LIN {X 0,Y 203.434,Z 438.559,A -85,B 0,C 180,E1 -21715.309,E2 -21715.309} C_VEL
LIN {X 0,Y 205.387,Z 432.116,A -85,B 0,C 180,E1 -21716.674,E2 -21716.674} C_VEL
LIN {X 0,Y 207.361,Z 424.448,A -85,B 0,C 180,E1 -21718.015,E2 -21718.015} C_VEL
LIN {X 0,Y 209.258,Z 416.269,A -85,B 0,C 180,E1 -21719.141,E2 -21719.141} C_VEL
LIN {X 0,Y 210.873,Z 408.266,A -85,B 0,C 180,E1 -21719.994,E2 -21719.994} C_VEL
LIN {X 0,Y 212.446,Z 398.341,A -85,B 0,C 180,E1 -21720.77,E2 -21720.77} C_VEL
LIN {X 0,Y 213.416,Z 388.623,A -85,B 0,C 180,E1 -21721.297,E2 -21721.297} C_VEL
LIN {X 0,Y 214.643,Z 363.756,A -85,B 0,C 180,E1 -21722.215,E2 -21722.215} C_VEL
LIN {X 0,Y 212.631,Z 347.83,A -85,B 0,C 180,E1 -21723.396,E2 -21723.396} C_VEL
LIN {X 0,Y 207.609,Z 336.115,A -85,B 0,C 180,E1 -21725.154,E2 -21725.154} C_VEL
LIN {X 0,Y 202.459,Z 325.893,A -85,B 0,C 180,E1 -21727.022,E2 -21727.022} C_VEL
LIN {X 0,Y 199.408,Z 320.617,A -85,B 0,C 180,E1 -21728.178,E2 -21728.178} C_VEL
LIN {X 0,Y 196.695,Z 316.069,A -85,B 0,C 180,E1 -21729.25,E2 -21729.25} C_VEL
LIN {X 0,Y 194.085,Z 311.74,A -85,B 0,C 180,E1 -21730.35,E2 -21730.35} C_VEL
LIN {X 0,Y 193.924,Z 311.308,A -85,B 0,C 180,E1 -21730.442,E2 -21730.442} C_VEL
LIN {X 0,Y 192.535,Z 306.316,A -85,B 0,C 180,E1 -21734.415,E2 -21734.415} C_VEL
LIN {X 0,Y 192.513,Z 306.314,A -85,B 0,C 180,E1 -21740.051,E2 -21740.051} C_VEL
LIN {X 0,Y 192.556,Z 306.307,A -85,B 0,C 180,E1 -21744.27,E2 -21744.27} C_VEL
LIN {X 0,Y 192.603,Z 306.292,A -85,B 0,C 180,E1 -21747.059,E2 -21747.059} C_VEL
LIN {X 0,Y 192.66,Z 306.284,A -85,B 0,C 180,E1 -21751.691,E2 -21751.691} C_VEL
LIN {X 0,Y 192.68,Z 306.291,A -85,B 0,C 180,E1 -21756.345,E2 -21756.345} C_VEL
LIN {X 0,Y 192.726,Z 306.291,A -85,B 0,C 180,E1 -21761.459,E2 -21761.459} C_VEL
LIN {X 0,Y 192.756,Z 306.268,A -85,B 0,C 180,E1 -21765.213,E2 -21765.213} C_VEL
LIN {X 0,Y 192.94,Z 306.247,A -85,B 0,C 180,E1 -21769.567,E2 -21769.567} C_VEL
LIN {X 0,Y 193.035,Z 306.233,A -85,B 0,C 180,E1 -21771.626,E2 -21771.626} C_VEL
LIN {X 0,Y 193.254,Z 306.208,A -85,B 0,C 180,E1 -21777.916,E2 -21777.916} C_VEL
LIN {X 0,Y 193.436,Z 306.199,A -85,B 0,C 180,E1 -21780,E2 -21780} C_VEL
LIN {X 0,Y 192.956,Z 306.254,A -85,B 0,C 180,E1 -21784.178,E2 -21784.178} C_VEL
LIN {X 0,Y 193.019,Z 306.241,A -85,B 0,C 180,E1 -21788.375,E2 -21788.375} C_VEL
LIN {X 0,Y 192.795,Z 306.27,A -85,B 0,C 180,E1 -21792.634,E2 -21792.634} C_VEL
LIN {X 0,Y 192.751,Z 306.28,A -85,B 0,C 180,E1 -21796.96,E2 -21796.96} C_VEL
LIN {X 0,Y 192.646,Z 306.299,A -85,B 0,C 180,E1 -21801.256,E2 -21801.256} C_VEL
LIN {X 0,Y 193.578,Z 309.046,A -85,B 0,C 180,E1 -21801.778,E2 -21801.778} C_VEL
LIN {X 0,Y 196.018,Z 311.688,A -85,B 0,C 180,E1 -21802.74,E2 -21802.74} C_VEL
LIN {X 0,Y 198.027,Z 314.946,A -85,B 0,C 180,E1 -21803.55,E2 -21803.55} C_VEL
LIN {X 0,Y 199.444,Z 316.867,A -85,B 0,C 180,E1 -21804.08,E2 -21804.08} C_VEL
LIN {X 0,Y 204.639,Z 324.932,A -85,B 0,C 180,E1 -21805.977,E2 -21805.977} C_VEL
LIN {X 0,Y 208.254,Z 331.276,A -85,B 0,C 180,E1 -21807.222,E2 -21807.222} C_VEL
LIN {X 0,Y 213.52,Z 342.533,A -85,B 0,C 180,E1 -21809.009,E2 -21809.009} C_VEL
LIN {X 0,Y 215.53,Z 347.517,A -85,B 0,C 180,E1 -21809.689,E2 -21809.689} C_VEL
LIN {X 0,Y 213.587,Z 380.961,A -85,B 0,C 180,E1 -21810.874,E2 -21810.874} C_VEL
LIN {X 0,Y 212.575,Z 391.195,A -85,B 0,C 180,E1 -21811.488,E2 -21811.488} C_VEL
LIN {X 0,Y 210.726,Z 403.434,A -85,B 0,C 180,E1 -21812.62,E2 -21812.62} C_VEL
LIN {X 0,Y 209.023,Z 411.772,A -85,B 0,C 180,E1 -21813.68,E2 -21813.68} C_VEL
LIN {X 0,Y 207.002,Z 419.999,A -85,B 0,C 180,E1 -21815.01,E2 -21815.01} C_VEL
LIN {X 0,Y 204.74,Z 428.007,A -85,B 0,C 180,E1 -21816.644,E2 -21816.644} C_VEL
LIN {X 0,Y 202.714,Z 434.266,A -85,B 0,C 180,E1 -21818.206,E2 -21818.206} C_VEL
LIN {X 0,Y 200.305,Z 440.944,A -85,B 0,C 180,E1 -21820.261,E2 -21820.261} C_VEL
LIN {X 0,Y 198.095,Z 446.483,A -85,B 0,C 180,E1 -21822.383,E2 -21822.383} C_VEL
LIN {X 0,Y 196.474,Z 450.562,A -85,B 0,C 180,E1 -21824.325,E2 -21824.325} C_VEL
LIN {X 0,Y 194.661,Z 454.577,A -85,B 0,C 180,E1 -21826.69,E2 -21826.69} C_VEL
LIN {X 0,Y 193.231,Z 457.717,A -85,B 0,C 180,E1 -21829.106,E2 -21829.106} C_VEL
LIN {X 0,Y 192.017,Z 460.05,A -85,B 0,C 180,E1 -21831.523,E2 -21831.523} C_VEL
LIN {X 0,Y 191.113,Z 461.68,A -85,B 0,C 180,E1 -21834.002,E2 -21834.002} C_VEL
LIN {X 0,Y 190.483,Z 462.591,A -85,B 0,C 180,E1 -21836.398,E2 -21836.398} C_VEL
LIN {X 0,Y 190.065,Z 462.86,A -85,B 0,C 180,E1 -21838.825,E2 -21838.825} C_VEL
LIN {X 0,Y 189.849,Z 462.453,A -85,B 0,C 180,E1 -21841.234,E2 -21841.234} C_VEL
LIN {X 0,Y 189.868,Z 461.377,A -85,B 0,C 180,E1 -21843.63,E2 -21843.63} C_VEL
LIN {X 0,Y 190.373,Z 458.386,A -85,B 0,C 180,E1 -21847.358,E2 -21847.358} C_VEL
LIN {X 0,Y 190.828,Z 455.896,A -85,B 0,C 180,E1 -21849.521,E2 -21849.521} C_VEL
LIN {X 0,Y 191.651,Z 451.34,A -85,B 0,C 180,E1 -21852.449,E2 -21852.449} C_VEL
LIN {X 0,Y 192.454,Z 447.029,A -85,B 0,C 180,E1 -21854.648,E2 -21854.648} C_VEL
LIN {X 0,Y 193.564,Z 441.616,A -85,B 0,C 180,E1 -21856.884,E2 -21856.884} C_VEL
LIN {X 0,Y 194.915,Z 434.909,A -85,B 0,C 180,E1 -21859.12,E2 -21859.12} C_VEL
LIN {X 0,Y 196.196,Z 428.057,A -85,B 0,C 180,E1 -21860.984,E2 -21860.984} C_VEL
LIN {X 0,Y 197.546,Z 420.587,A -85,B 0,C 180,E1 -21862.641,E2 -21862.641} C_VEL
LIN {X 0,Y 198.959,Z 412.007,A -85,B 0,C 180,E1 -21864.171,E2 -21864.171} C_VEL
LIN {X 0,Y 200.337,Z 401.733,A -85,B 0,C 180,E1 -21865.599,E2 -21865.599} C_VEL
LIN {X 0,Y 201.427,Z 390.601,A -85,B 0,C 180,E1 -21866.687,E2 -21866.687} C_VEL
LIN {X 0,Y 202.147,Z 380.872,A -85,B 0,C 180,E1 -21867.322,E2 -21867.322} C_VEL
LIN {X 0,Y 203.703,Z 338.888,A -85,B 0,C 180,E1 -21868.912,E2 -21868.912} C_VEL
LIN {X 0,Y 202.454,Z 331.462,A -85,B 0,C 180,E1 -21869.352,E2 -21869.352} C_VEL
LIN {X 0,Y 196.567,Z 313.956,A -85,B 0,C 180,E1 -21870.782,E2 -21870.782} C_VEL
LIN {X 0,Y 193.402,Z 306.719,A -85,B 0,C 180,E1 -21871.497,E2 -21871.497} C_VEL
LIN {X 0,Y 193.304,Z 306.221,A -85,B 0,C 180,E1 -21871.615,E2 -21871.615} C_VEL
LIN {X 0,Y 193.033,Z 306.255,A -85,B 0,C 180,E1 -21878.374,E2 -21878.374} C_VEL
LIN {X 0,Y 192.798,Z 306.271,A -85,B 0,C 180,E1 -21882.633,E2 -21882.633} C_VEL
LIN {X 0,Y 192.749,Z 306.286,A -85,B 0,C 180,E1 -21886.959,E2 -21886.959} C_VEL
LIN {X 0,Y 192.609,Z 306.28,A -85,B 0,C 180,E1 -21891.4,E2 -21891.4} C_VEL
LIN {X 0,Y 192.648,Z 306.291,A -85,B 0,C 180,E1 -21894.212,E2 -21894.212} C_VEL
LIN {X 0,Y 192.65,Z 306.305,A -85,B 0,C 180,E1 -21898.891,E2 -21898.891} C_VEL
LIN {X 0,Y 192.598,Z 306.3,A -85,B 0,C 180,E1 -21903.185,E2 -21903.185} C_VEL
LIN {X 0,Y 192.551,Z 306.312,A -85,B 0,C 180,E1 -21908.351,E2 -21908.351} C_VEL
LIN {X 0,Y 192.537,Z 306.306,A -85,B 0,C 180,E1 -21913.909,E2 -21913.909} C_VEL
LIN {X 0,Y 192.576,Z 306.308,A -85,B 0,C 180,E1 -21918.935,E2 -21918.935} C_VEL
LIN {X 0,Y 192.616,Z 306.291,A -85,B 0,C 180,E1 -21923.388,E2 -21923.388} C_VEL
LIN {X 0,Y 192.604,Z 306.294,A -85,B 0,C 180,E1 -21927.059,E2 -21927.059} C_VEL
LIN {X 0,Y 192.661,Z 306.298,A -85,B 0,C 180,E1 -21931.691,E2 -21931.691} C_VEL
LIN {X 0,Y 192.702,Z 306.283,A -85,B 0,C 180,E1 -21936.348,E2 -21936.348} C_VEL
LIN {X 0,Y 192.728,Z 306.276,A -85,B 0,C 180,E1 -21941.457,E2 -21941.457} C_VEL
LIN {X 0,Y 192.758,Z 306.285,A -85,B 0,C 180,E1 -21945.213,E2 -21945.213} C_VEL
LIN {X 0,Y 192.941,Z 306.26,A -85,B 0,C 180,E1 -21949.566,E2 -21949.566} C_VEL
LIN {X 0,Y 192.978,Z 306.24,A -85,B 0,C 180,E1 -21953.727,E2 -21953.727} C_VEL
LIN {X 0,Y 193.255,Z 306.214,A -85,B 0,C 180,E1 -21957.916,E2 -21957.916} C_VEL
LIN {X 0,Y 193.436,Z 306.198,A -85,B 0,C 180,E1 -21960,E2 -21960} C_VEL
LIN {X 0,Y 192.964,Z 306.258,A -85,B 0,C 180,E1 -21964.177,E2 -21964.177} C_VEL
LIN {X 0,Y 193.03,Z 306.237,A -85,B 0,C 180,E1 -21968.374,E2 -21968.374} C_VEL
LIN {X 0,Y 192.795,Z 306.275,A -85,B 0,C 180,E1 -21972.634,E2 -21972.634} C_VEL
LIN {X 0,Y 192.75,Z 306.286,A -85,B 0,C 180,E1 -21976.959,E2 -21976.959} C_VEL
LIN {X 0,Y 192.61,Z 306.292,A -85,B 0,C 180,E1 -21981.4,E2 -21981.4} C_VEL
LIN {X 0,Y 192.642,Z 306.3,A -85,B 0,C 180,E1 -21984.213,E2 -21984.213} C_VEL
LIN {X 0,Y 192.639,Z 306.296,A -85,B 0,C 180,E1 -21988.889,E2 -21988.889} C_VEL
LIN {X 0,Y 192.592,Z 306.307,A -85,B 0,C 180,E1 -21993.187,E2 -21993.187} C_VEL
LIN {X 0,Y 192.547,Z 306.303,A -85,B 0,C 180,E1 -21998.353,E2 -21998.353} C_VEL
LIN {X 0,Y 192.488,Z 306.311,A -85,B 0,C 180,E1 -22003.096,E2 -22003.096} C_VEL
LIN {X 0,Y 192.489,Z 306.32,A -85,B 0,C 180,E1 -22006.905,E2 -22006.905} C_VEL
LIN {X 0,Y 192.549,Z 306.312,A -85,B 0,C 180,E1 -22011.649,E2 -22011.649} C_VEL
LIN {X 0,Y 192.654,Z 306.48,A -85,B 0,C 180,E1 -22016.513,E2 -22016.513} C_VEL
LIN {X 0,Y 194.109,Z 313.398,A -85,B 0,C 180,E1 -22020.468,E2 -22020.468} C_VEL
LIN {X 0,Y 199.249,Z 328.764,A -85,B 0,C 180,E1 -22021.772,E2 -22021.772} C_VEL
LIN {X 0,Y 203.033,Z 359.935,A -85,B 0,C 180,E1 -22023.469,E2 -22023.469} C_VEL
LIN {X 0,Y 202.374,Z 380.986,A -85,B 0,C 180,E1 -22024.245,E2 -22024.245} C_VEL
LIN {X 0,Y 201.379,Z 386.811,A -85,B 0,C 180,E1 -22024.384,E2 -22024.384} C_VEL
LIN {X 0,Y 197.854,Z 396.121,A -85,B 0,C 180,E1 -22024.575,E2 -22024.575} C_VEL
LIN {X 0,Y 194.572,Z 404.335,A -85,B 0,C 180,E1 -22024.961,E2 -22024.961} C_VEL
LIN {X 0,Y 193.494,Z 408.938,A -85,B 0,C 180,E1 -22025.38,E2 -22025.38} C_VEL
LIN {X 0,Y 193.28,Z 410.781,A -85,B 0,C 180,E1 -22025.582,E2 -22025.582} C_VEL
LIN {X 0,Y 191.835,Z 421.682,A -85,B 0,C 180,E1 -22027.093,E2 -22027.093} C_VEL
LIN {X 0,Y 190.225,Z 430.12,A -85,B 0,C 180,E1 -22028.603,E2 -22028.603} C_VEL
LIN {X 0,Y 189.015,Z 437.111,A -85,B 0,C 180,E1 -22030.167,E2 -22030.167} C_VEL
LIN {X 0,Y 187.632,Z 443.888,A -85,B 0,C 180,E1 -22032.001,E2 -22032.001} C_VEL
LIN {X 0,Y 186.264,Z 450.309,A -85,B 0,C 180,E1 -22034.125,E2 -22034.125} C_VEL
LIN {X 0,Y 185.196,Z 455.643,A -85,B 0,C 180,E1 -22036.28,E2 -22036.28} C_VEL
LIN {X 0,Y 184.197,Z 461.047,A -85,B 0,C 180,E1 -22039.002,E2 -22039.002} C_VEL
LIN {X 0,Y 183.657,Z 464.529,A -85,B 0,C 180,E1 -22041.195,E2 -22041.195} C_VEL
LIN {X 0,Y 183.178,Z 468.522,A -85,B 0,C 180,E1 -22044.496,E2 -22044.496} C_VEL
LIN {X 0,Y 183.099,Z 471.231,A -85,B 0,C 180,E1 -22047.8,E2 -22047.8} C_VEL
LIN {X 0,Y 183.2,Z 472.28,A -85,B 0,C 180,E1 -22050,E2 -22050} C_VEL
LIN {X 0,Y 183.052,Z 472.991,A -85,B 0,C 180,E1 -22053.412,E2 -22053.412} C_VEL
LIN {X 0,Y 183.303,Z 472.546,A -85,B 0,C 180,E1 -22056.605,E2 -22056.605} C_VEL
LIN {X 0,Y 183.684,Z 471.57,A -85,B 0,C 180,E1 -22058.803,E2 -22058.803} C_VEL
LIN {X 0,Y 184.348,Z 470.105,A -85,B 0,C 180,E1 -22060.988,E2 -22060.988} C_VEL
LIN {X 0,Y 185.765,Z 466.977,A -85,B 0,C 180,E1 -22064.235,E2 -22064.235} C_VEL
LIN {X 0,Y 187.76,Z 462.559,A -85,B 0,C 180,E1 -22067.424,E2 -22067.424} C_VEL
LIN {X 0,Y 190.383,Z 456.487,A -85,B 0,C 180,E1 -22070.529,E2 -22070.529} C_VEL
LIN {X 0,Y 192.486,Z 451.491,A -85,B 0,C 180,E1 -22072.542,E2 -22072.542} C_VEL
LIN {X 0,Y 194.842,Z 445.491,A -85,B 0,C 180,E1 -22074.506,E2 -22074.506} C_VEL
LIN {X 0,Y 197.684,Z 437.209,A -85,B 0,C 180,E1 -22076.668,E2 -22076.668} C_VEL
LIN {X 0,Y 200.136,Z 429.569,A -85,B 0,C 180,E1 -22078.223,E2 -22078.223} C_VEL
LIN {X 0,Y 202.757,Z 419.419,A -85,B 0,C 180,E1 -22079.884,E2 -22079.884} C_VEL
LIN {X 0,Y 205.191,Z 408.083,A -85,B 0,C 180,E1 -22081.169,E2 -22081.169} C_VEL
LIN {X 0,Y 206.761,Z 398.675,A -85,B 0,C 180,E1 -22081.926,E2 -22081.926} C_VEL
LIN {X 0,Y 207.771,Z 389.397,A -85,B 0,C 180,E1 -22082.455,E2 -22082.455} C_VEL
LIN {X 0,Y 209.142,Z 364.971,A -85,B 0,C 180,E1 -22083.377,E2 -22083.377} C_VEL
LIN {X 0,Y 207.395,Z 350.739,A -85,B 0,C 180,E1 -22084.481,E2 -22084.481} C_VEL
LIN {X 0,Y 202.339,Z 338.752,A -85,B 0,C 180,E1 -22086.372,E2 -22086.372} C_VEL
LIN {X 0,Y 197.56,Z 329.355,A -85,B 0,C 180,E1 -22088.242,E2 -22088.242} C_VEL
LIN {X 0,Y 192.786,Z 321.063,A -85,B 0,C 180,E1 -22090.214,E2 -22090.214} C_VEL
LIN {X 0,Y 189.733,Z 316.142,A -85,B 0,C 180,E1 -22091.572,E2 -22091.572} C_VEL
LIN {X 0,Y 186.926,Z 311.969,A -85,B 0,C 180,E1 -22092.874,E2 -22092.874} C_VEL
LIN {X 0,Y 186.457,Z 310.795,A -85,B 0,C 180,E1 -22093.256,E2 -22093.256} C_VEL
LIN {X 0,Y 185.446,Z 307.2,A -85,B 0,C 180,E1 -22096.504,E2 -22096.504} C_VEL
LIN {X 0,Y 185.463,Z 307.191,A -85,B 0,C 180,E1 -22099.894,E2 -22099.894} C_VEL
LIN {X 0,Y 185.502,Z 307.179,A -85,B 0,C 180,E1 -22102.711,E2 -22102.711} C_VEL
LIN {X 0,Y 185.539,Z 307.172,A -85,B 0,C 180,E1 -22107.974,E2 -22107.974} C_VEL
LIN {X 0,Y 185.577,Z 307.178,A -85,B 0,C 180,E1 -22110.576,E2 -22110.576} C_VEL
LIN {X 0,Y 185.575,Z 307.181,A -85,B 0,C 180,E1 -22115.381,E2 -22115.381} C_VEL
LIN {X 0,Y 185.668,Z 307.17,A -85,B 0,C 180,E1 -22121.135,E2 -22121.135} C_VEL
LIN {X 0,Y 185.688,Z 307.146,A -85,B 0,C 180,E1 -22124.637,E2 -22124.637} C_VEL
LIN {X 0,Y 185.884,Z 307.126,A -85,B 0,C 180,E1 -22129.417,E2 -22129.417} C_VEL
LIN {X 0,Y 185.944,Z 307.133,A -85,B 0,C 180,E1 -22133.49,E2 -22133.49} C_VEL
LIN {X 0,Y 186.198,Z 307.086,A -85,B 0,C 180,E1 -22137.837,E2 -22137.837} C_VEL
LIN {X 0,Y 186.399,Z 307.076,A -85,B 0,C 180,E1 -22140,E2 -22140} C_VEL
LIN {X 0,Y 185.903,Z 307.134,A -85,B 0,C 180,E1 -22144.337,E2 -22144.337} C_VEL
LIN {X 0,Y 185.968,Z 307.12,A -85,B 0,C 180,E1 -22148.695,E2 -22148.695} C_VEL
LIN {X 0,Y 185.722,Z 307.152,A -85,B 0,C 180,E1 -22153.124,E2 -22153.124} C_VEL
LIN {X 0,Y 185.689,Z 307.236,A -85,B 0,C 180,E1 -22158.793,E2 -22158.793} C_VEL
LIN {X 0,Y 186.476,Z 309.725,A -85,B 0,C 180,E1 -22159.265,E2 -22159.265} C_VEL
LIN {X 0,Y 188.492,Z 312.038,A -85,B 0,C 180,E1 -22160.175,E2 -22160.175} C_VEL
LIN {X 0,Y 189.26,Z 312.966,A -85,B 0,C 180,E1 -22160.515,E2 -22160.515} C_VEL
LIN {X 0,Y 191.39,Z 316.203,A -85,B 0,C 180,E1 -22161.473,E2 -22161.473} C_VEL
LIN {X 0,Y 192.579,Z 317.611,A -85,B 0,C 180,E1 -22161.967,E2 -22161.967} C_VEL
LIN {X 0,Y 198.035,Z 325.775,A -85,B 0,C 180,E1 -22164.157,E2 -22164.157} C_VEL
LIN {X 0,Y 202.881,Z 333.982,A -85,B 0,C 180,E1 -22165.978,E2 -22165.978} C_VEL
LIN {X 0,Y 207.643,Z 343.937,A -85,B 0,C 180,E1 -22167.699,E2 -22167.699} C_VEL
LIN {X 0,Y 209.982,Z 349.731,A -85,B 0,C 180,E1 -22168.539,E2 -22168.539} C_VEL
LIN {X 0,Y 208.007,Z 381.708,A -85,B 0,C 180,E1 -22169.704,E2 -22169.704} C_VEL
LIN {X 0,Y 206.773,Z 392.837,A -85,B 0,C 180,E1 -22170.398,E2 -22170.398} C_VEL
LIN {X 0,Y 204.99,Z 403.83,A -85,B 0,C 180,E1 -22171.482,E2 -22171.482} C_VEL
LIN {X 0,Y 203.224,Z 412.033,A -85,B 0,C 180,E1 -22172.55,E2 -22172.55} C_VEL
LIN {X 0,Y 200.862,Z 420.979,A -85,B 0,C 180,E1 -22174.044,E2 -22174.044} C_VEL
LIN {X 0,Y 198.724,Z 428.205,A -85,B 0,C 180,E1 -22175.572,E2 -22175.572} C_VEL
LIN {X 0,Y 196.122,Z 435.719,A -85,B 0,C 180,E1 -22177.531,E2 -22177.531} C_VEL
LIN {X 0,Y 193.702,Z 441.948,A -85,B 0,C 180,E1 -22179.558,E2 -22179.558} C_VEL
LIN {X 0,Y 190.717,Z 449.06,A -85,B 0,C 180,E1 -22182.525,E2 -22182.525} C_VEL
LIN {X 0,Y 188.712,Z 453.553,A -85,B 0,C 180,E1 -22185.04,E2 -22185.04} C_VEL
LIN {X 0,Y 187.023,Z 456.907,A -85,B 0,C 180,E1 -22187.438,E2 -22187.438} C_VEL
LIN {X 0,Y 185.64,Z 459.533,A -85,B 0,C 180,E1 -22189.941,E2 -22189.941} C_VEL
LIN {X 0,Y 184.259,Z 461.783,A -85,B 0,C 180,E1 -22193.224,E2 -22193.224} C_VEL
LIN {X 0,Y 183.703,Z 462.53,A -85,B 0,C 180,E1 -22194.981,E2 -22194.981} C_VEL
LIN {X 0,Y 183.15,Z 463.007,A -85,B 0,C 180,E1 -22197.587,E2 -22197.587} C_VEL
LIN {X 0,Y 182.842,Z 462.818,A -85,B 0,C 180,E1 -22200.022,E2 -22200.022} C_VEL
LIN {X 0,Y 182.759,Z 462.008,A -85,B 0,C 180,E1 -22202.52,E2 -22202.52} C_VEL
LIN {X 0,Y 182.882,Z 460.569,A -85,B 0,C 180,E1 -22204.994,E2 -22204.994} C_VEL
LIN {X 0,Y 183.297,Z 458.47,A -85,B 0,C 180,E1 -22207.455,E2 -22207.455} C_VEL
LIN {X 0,Y 183.812,Z 455.703,A -85,B 0,C 180,E1 -22209.873,E2 -22209.873} C_VEL
LIN {X 0,Y 184.666,Z 451.157,A -85,B 0,C 180,E1 -22212.846,E2 -22212.846} C_VEL
LIN {X 0,Y 185.52,Z 446.633,A -85,B 0,C 180,E1 -22215.185,E2 -22215.185} C_VEL
LIN {X 0,Y 186.924,Z 440.18,A -85,B 0,C 180,E1 -22217.838,E2 -22217.838} C_VEL
LIN {X 0,Y 188.118,Z 434.356,A -85,B 0,C 180,E1 -22219.779,E2 -22219.779} C_VEL
LIN {X 0,Y 189.743,Z 426.108,A -85,B 0,C 180,E1 -22222.017,E2 -22222.017} C_VEL
LIN {X 0,Y 191.66,Z 415.505,A -85,B 0,C 180,E1 -22224.213,E2 -22224.213} C_VEL
LIN {X 0,Y 192.934,Z 407.016,A -85,B 0,C 180,E1 -22225.561,E2 -22225.561} C_VEL
LIN {X 0,Y 193.927,Z 398.525,A -85,B 0,C 180,E1 -22226.624,E2 -22226.624} C_VEL
LIN {X 0,Y 194.881,Z 389.268,A -85,B 0,C 180,E1 -22227.481,E2 -22227.481} C_VEL
LIN {X 0,Y 195.524,Z 379.672,A -85,B 0,C 180,E1 -22228.095,E2 -22228.095} C_VEL
LIN {X 0,Y 197.062,Z 339.354,A -85,B 0,C 180,E1 -22229.655,E2 -22229.655} C_VEL
LIN {X 0,Y 195.953,Z 333.197,A -85,B 0,C 180,E1 -22230.048,E2 -22230.048} C_VEL
LIN {X 0,Y 190.398,Z 316.71,A -85,B 0,C 180,E1 -22231.457,E2 -22231.457} C_VEL
LIN {X 0,Y 186.2,Z 307.493,A -85,B 0,C 180,E1 -22232.434,E2 -22232.434} C_VEL
LIN {X 0,Y 186.119,Z 307.113,A -85,B 0,C 180,E1 -22232.57,E2 -22232.57} C_VEL
LIN {X 0,Y 185.981,Z 307.132,A -85,B 0,C 180,E1 -22238.694,E2 -22238.694} C_VEL
LIN {X 0,Y 185.725,Z 307.153,A -85,B 0,C 180,E1 -22243.123,E2 -22243.123} C_VEL
LIN {X 0,Y 185.685,Z 307.165,A -85,B 0,C 180,E1 -22247.625,E2 -22247.625} C_VEL
LIN {X 0,Y 185.574,Z 307.156,A -85,B 0,C 180,E1 -22252.254,E2 -22252.254} C_VEL
LIN {X 0,Y 185.561,Z 307.187,A -85,B 0,C 180,E1 -22257.031,E2 -22257.031} C_VEL
LIN {X 0,Y 185.579,Z 307.183,A -85,B 0,C 180,E1 -22259.492,E2 -22259.492} C_VEL
LIN {X 0,Y 185.499,Z 307.187,A -85,B 0,C 180,E1 -22264.631,E2 -22264.631} C_VEL
LIN {X 0,Y 185.505,Z 307.193,A -85,B 0,C 180,E1 -22267.312,E2 -22267.312} C_VEL
LIN {X 0,Y 185.473,Z 307.189,A -85,B 0,C 180,E1 -22270.725,E2 -22270.725} C_VEL
LIN {X 0,Y 185.528,Z 307.185,A -85,B 0,C 180,E1 -22276.031,E2 -22276.031} C_VEL
LIN {X 0,Y 185.536,Z 307.184,A -85,B 0,C 180,E1 -22279.913,E2 -22279.913} C_VEL
LIN {X 0,Y 185.557,Z 307.172,A -85,B 0,C 180,E1 -22282.699,E2 -22282.699} C_VEL
LIN {X 0,Y 185.542,Z 307.178,A -85,B 0,C 180,E1 -22287.974,E2 -22287.974} C_VEL
LIN {X 0,Y 185.579,Z 307.179,A -85,B 0,C 180,E1 -22290.575,E2 -22290.575} C_VEL
LIN {X 0,Y 185.583,Z 307.173,A -85,B 0,C 180,E1 -22295.382,E2 -22295.382} C_VEL
LIN {X 0,Y 185.671,Z 307.155,A -85,B 0,C 180,E1 -22301.133,E2 -22301.133} C_VEL
LIN {X 0,Y 185.689,Z 307.165,A -85,B 0,C 180,E1 -22304.636,E2 -22304.636} C_VEL
LIN {X 0,Y 185.884,Z 307.139,A -85,B 0,C 180,E1 -22309.417,E2 -22309.417} C_VEL
LIN {X 0,Y 185.941,Z 307.116,A -85,B 0,C 180,E1 -22313.489,E2 -22313.489} C_VEL
LIN {X 0,Y 186.199,Z 307.093,A -85,B 0,C 180,E1 -22317.837,E2 -22317.837} C_VEL
LIN {X 0,Y 186.4,Z 307.074,A -85,B 0,C 180,E1 -22320,E2 -22320} C_VEL
LIN {X 0,Y 185.911,Z 307.136,A -85,B 0,C 180,E1 -22324.336,E2 -22324.336} C_VEL
LIN {X 0,Y 185.977,Z 307.115,A -85,B 0,C 180,E1 -22328.694,E2 -22328.694} C_VEL
LIN {X 0,Y 185.723,Z 307.157,A -85,B 0,C 180,E1 -22333.123,E2 -22333.123} C_VEL
LIN {X 0,Y 185.683,Z 307.167,A -85,B 0,C 180,E1 -22337.625,E2 -22337.625} C_VEL
LIN {X 0,Y 185.572,Z 307.172,A -85,B 0,C 180,E1 -22342.254,E2 -22342.254} C_VEL
LIN {X 0,Y 185.554,Z 307.183,A -85,B 0,C 180,E1 -22347.033,E2 -22347.033} C_VEL
LIN {X 0,Y 185.573,Z 307.177,A -85,B 0,C 180,E1 -22349.494,E2 -22349.494} C_VEL
LIN {X 0,Y 185.495,Z 307.193,A -85,B 0,C 180,E1 -22354.633,E2 -22354.633} C_VEL
LIN {X 0,Y 185.502,Z 307.186,A -85,B 0,C 180,E1 -22357.314,E2 -22357.314} C_VEL
LIN {X 0,Y 185.467,Z 307.173,A -85,B 0,C 180,E1 -22360.725,E2 -22360.725} C_VEL
LIN {X 0,Y 185.458,Z 307.195,A -85,B 0,C 180,E1 -22366.055,E2 -22366.055} C_VEL
LIN {X 0,Y 185.465,Z 307.194,A -85,B 0,C 180,E1 -22369.896,E2 -22369.896} C_VEL
LIN {X 0,Y 185.504,Z 307.188,A -85,B 0,C 180,E1 -22372.712,E2 -22372.712} C_VEL
LIN {X 0,Y 185.599,Z 307.344,A -85,B 0,C 180,E1 -22376.001,E2 -22376.001} C_VEL
LIN {X 0,Y 186.818,Z 313.253,A -85,B 0,C 180,E1 -22379.525,E2 -22379.525} C_VEL
LIN {X 0,Y 192.764,Z 330.38,A -85,B 0,C 180,E1 -22381.047,E2 -22381.047} C_VEL
LIN {X 0,Y 196.469,Z 361.488,A -85,B 0,C 180,E1 -22382.81,E2 -22382.81} C_VEL
LIN {X 0,Y 195.25,Z 390.957,A -85,B 0,C 180,E1 -22383.972,E2 -22383.972} C_VEL
LIN {X 0,Y 194.486,Z 400.625,A -85,B 0,C 180,E1 -22384.609,E2 -22384.609} C_VEL
LIN {X 0,Y 193.28,Z 410.781,A -85,B 0,C 180,E1 -22385.582,E2 -22385.582} C_VEL
LIN {X 0,Y 192.111,Z 416.18,A -85,B 0,C 180,E1 -22386.193,E2 -22386.193} C_VEL
LIN {X 0,Y 189.902,Z 421.303,A -85,B 0,C 180,E1 -22386.805,E2 -22386.805} C_VEL
LIN {X 0,Y 184.59,Z 430.867,A -85,B 0,C 180,E1 -22388.279,E2 -22388.279} C_VEL
LIN {X 0,Y 182.575,Z 435.503,A -85,B 0,C 180,E1 -22389.268,E2 -22389.268} C_VEL
LIN {X 0,Y 182.148,Z 436.983,A -85,B 0,C 180,E1 -22389.647,E2 -22389.647} C_VEL
LIN {X 0,Y 180.875,Z 442.987,A -85,B 0,C 180,E1 -22391.304,E2 -22391.304} C_VEL
LIN {X 0,Y 179.428,Z 449.523,A -85,B 0,C 180,E1 -22393.503,E2 -22393.503} C_VEL
LIN {X 0,Y 178.292,Z 454.958,A -85,B 0,C 180,E1 -22395.738,E2 -22395.738} C_VEL
LIN {X 0,Y 177.209,Z 460.451,A -85,B 0,C 180,E1 -22398.563,E2 -22398.563} C_VEL
LIN {X 0,Y 176.627,Z 464.014,A -85,B 0,C 180,E1 -22400.842,E2 -22400.842} C_VEL
LIN {X 0,Y 176.11,Z 468.082,A -85,B 0,C 180,E1 -22404.274,E2 -22404.274} C_VEL
LIN {X 0,Y 175.989,Z 470.154,A -85,B 0,C 180,E1 -22406.709,E2 -22406.709} C_VEL
LIN {X 0,Y 176.105,Z 471.979,A -85,B 0,C 180,E1 -22410,E2 -22410} C_VEL
LIN {X 0,Y 175.953,Z 472.7,A -85,B 0,C 180,E1 -22413.077,E2 -22413.077} C_VEL
LIN {X 0,Y 176.243,Z 472.404,A -85,B 0,C 180,E1 -22416.87,E2 -22416.87} C_VEL
LIN {X 0,Y 176.657,Z 471.477,A -85,B 0,C 180,E1 -22419.156,E2 -22419.156} C_VEL
LIN {X 0,Y 177.361,Z 470.084,A -85,B 0,C 180,E1 -22421.427,E2 -22421.427} C_VEL
LIN {X 0,Y 178.889,Z 467.03,A -85,B 0,C 180,E1 -22424.795,E2 -22424.795} C_VEL
LIN {X 0,Y 180.989,Z 462.721,A -85,B 0,C 180,E1 -22428.098,E2 -22428.098} C_VEL
LIN {X 0,Y 183.765,Z 456.804,A -85,B 0,C 180,E1 -22431.304,E2 -22431.304} C_VEL
LIN {X 0,Y 186.511,Z 450.517,A -85,B 0,C 180,E1 -22433.895,E2 -22433.895} C_VEL
LIN {X 0,Y 189.085,Z 444.378,A -85,B 0,C 180,E1 -22435.895,E2 -22435.895} C_VEL
LIN {X 0,Y 191.416,Z 437.969,A -85,B 0,C 180,E1 -22437.615,E2 -22437.615} C_VEL
LIN {X 0,Y 194.289,Z 429.425,A -85,B 0,C 180,E1 -22439.426,E2 -22439.426} C_VEL
LIN {X 0,Y 196.695,Z 420.661,A -85,B 0,C 180,E1 -22440.904,E2 -22440.904} C_VEL
LIN {X 0,Y 199.465,Z 408.835,A -85,B 0,C 180,E1 -22442.336,E2 -22442.336} C_VEL
LIN {X 0,Y 201.227,Z 398.833,A -85,B 0,C 180,E1 -22443.166,E2 -22443.166} C_VEL
LIN {X 0,Y 202.264,Z 389.942,A -85,B 0,C 180,E1 -22443.694,E2 -22443.694} C_VEL
LIN {X 0,Y 203.687,Z 365.642,A -85,B 0,C 180,E1 -22444.644,E2 -22444.644} C_VEL
LIN {X 0,Y 202.263,Z 353.686,A -85,B 0,C 180,E1 -22445.614,E2 -22445.614} C_VEL
LIN {X 0,Y 197.931,Z 343.059,A -85,B 0,C 180,E1 -22447.372,E2 -22447.372} C_VEL
LIN {X 0,Y 192.277,Z 331.715,A -85,B 0,C 180,E1 -22449.74,E2 -22449.74} C_VEL
LIN {X 0,Y 188.721,Z 325.73,A -85,B 0,C 180,E1 -22451.326,E2 -22451.326} C_VEL
LIN {X 0,Y 185.913,Z 321.155,A -85,B 0,C 180,E1 -22452.653,E2 -22452.653} C_VEL
LIN {X 0,Y 182.488,Z 315.869,A -85,B 0,C 180,E1 -22454.367,E2 -22454.367} C_VEL
LIN {X 0,Y 179.527,Z 311.542,A -85,B 0,C 180,E1 -22455.984,E2 -22455.984} C_VEL
LIN {X 0,Y 179.104,Z 310.487,A -85,B 0,C 180,E1 -22456.34,E2 -22456.34} C_VEL
LIN {X 0,Y 178.421,Z 308.065,A -85,B 0,C 180,E1 -22458.865,E2 -22458.865} C_VEL
LIN {X 0,Y 178.418,Z 308.064,A -85,B 0,C 180,E1 -22463.782,E2 -22463.782} C_VEL
LIN {X 0,Y 178.481,Z 308.053,A -85,B 0,C 180,E1 -22466.546,E2 -22466.546} C_VEL
LIN {X 0,Y 178.518,Z 308.061,A -85,B 0,C 180,E1 -22470.006,E2 -22470.006} C_VEL
LIN {X 0,Y 178.515,Z 308.058,A -85,B 0,C 180,E1 -22474.886,E2 -22474.886} C_VEL
LIN {X 0,Y 178.616,Z 308.046,A -85,B 0,C 180,E1 -22480.786,E2 -22480.786} C_VEL
LIN {X 0,Y 178.651,Z 308.034,A -85,B 0,C 180,E1 -22486.348,E2 -22486.348} C_VEL
LIN {X 0,Y 178.908,Z 307.989,A -85,B 0,C 180,E1 -22490.96,E2 -22490.96} C_VEL
LIN {X 0,Y 178.858,Z 308,A -85,B 0,C 180,E1 -22495.493,E2 -22495.493} C_VEL
LIN {X 0,Y 179.363,Z 307.952,A -85,B 0,C 180,E1 -22500,E2 -22500} C_VEL
LIN {X 0,Y 178.85,Z 308.014,A -85,B 0,C 180,E1 -22504.508,E2 -22504.508} C_VEL
LIN {X 0,Y 178.899,Z 308.003,A -85,B 0,C 180,E1 -22509.041,E2 -22509.041} C_VEL
LIN {X 0,Y 178.633,Z 308.049,A -85,B 0,C 180,E1 -22514.817,E2 -22514.817} C_VEL
LIN {X 0,Y 178.625,Z 308.042,A -85,B 0,C 180,E1 -22515.767,E2 -22515.767} C_VEL
LIN {X 0,Y 179.529,Z 310.76,A -85,B 0,C 180,E1 -22516.415,E2 -22516.415} C_VEL
LIN {X 0,Y 181.521,Z 312.92,A -85,B 0,C 180,E1 -22517.461,E2 -22517.461} C_VEL
LIN {X 0,Y 182.387,Z 313.597,A -85,B 0,C 180,E1 -22517.883,E2 -22517.883} C_VEL
LIN {X 0,Y 184.268,Z 316.842,A -85,B 0,C 180,E1 -22518.883,E2 -22518.883} C_VEL
LIN {X 0,Y 185.987,Z 318.787,A -85,B 0,C 180,E1 -22519.679,E2 -22519.679} C_VEL
LIN {X 0,Y 188.59,Z 322.441,A -85,B 0,C 180,E1 -22520.877,E2 -22520.877} C_VEL
LIN {X 0,Y 194.026,Z 330.695,A -85,B 0,C 180,E1 -22523.216,E2 -22523.216} C_VEL
LIN {X 0,Y 198.595,Z 338.507,A -85,B 0,C 180,E1 -22525.025,E2 -22525.025} C_VEL
LIN {X 0,Y 203.38,Z 349.007,A -85,B 0,C 180,E1 -22526.893,E2 -22526.893} C_VEL
LIN {X 0,Y 204.511,Z 351.786,A -85,B 0,C 180,E1 -22527.32,E2 -22527.32} C_VEL
LIN {X 0,Y 202.578,Z 381.818,A -85,B 0,C 180,E1 -22528.438,E2 -22528.438} C_VEL
LIN {X 0,Y 201.319,Z 392.753,A -85,B 0,C 180,E1 -22529.128,E2 -22529.128} C_VEL
LIN {X 0,Y 199.348,Z 404.198,A -85,B 0,C 180,E1 -22530.263,E2 -22530.263} C_VEL
LIN {X 0,Y 197.187,Z 413.568,A -85,B 0,C 180,E1 -22531.539,E2 -22531.539} C_VEL
LIN {X 0,Y 194.993,Z 421.421,A -85,B 0,C 180,E1 -22532.9,E2 -22532.9} C_VEL
LIN {X 0,Y 192.776,Z 428.493,A -85,B 0,C 180,E1 -22534.431,E2 -22534.431} C_VEL
LIN {X 0,Y 190.293,Z 435.277,A -85,B 0,C 180,E1 -22536.223,E2 -22536.223} C_VEL
LIN {X 0,Y 187.804,Z 441.351,A -85,B 0,C 180,E1 -22538.202,E2 -22538.202} C_VEL
LIN {X 0,Y 185.165,Z 447.263,A -85,B 0,C 180,E1 -22540.617,E2 -22540.617} C_VEL
LIN {X 0,Y 182.318,Z 453.436,A -85,B 0,C 180,E1 -22543.937,E2 -22543.937} C_VEL
LIN {X 0,Y 180.134,Z 457.442,A -85,B 0,C 180,E1 -22546.943,E2 -22546.943} C_VEL
LIN {X 0,Y 178.69,Z 459.986,A -85,B 0,C 180,E1 -22549.539,E2 -22549.539} C_VEL
LIN {X 0,Y 177.049,Z 462.328,A -85,B 0,C 180,E1 -22553.458,E2 -22553.458} C_VEL
LIN {X 0,Y 176.165,Z 463.178,A -85,B 0,C 180,E1 -22556.907,E2 -22556.907} C_VEL
LIN {X 0,Y 175.867,Z 463.173,A -85,B 0,C 180,E1 -22558.702,E2 -22558.702} C_VEL
LIN {X 0,Y 175.68,Z 462.484,A -85,B 0,C 180,E1 -22561.655,E2 -22561.655} C_VEL
LIN {X 0,Y 175.688,Z 461.458,A -85,B 0,C 180,E1 -22563.895,E2 -22563.895} C_VEL
LIN {X 0,Y 176.039,Z 459.424,A -85,B 0,C 180,E1 -22566.669,E2 -22566.669} C_VEL
LIN {X 0,Y 176.789,Z 455.481,A -85,B 0,C 180,E1 -22570.251,E2 -22570.251} C_VEL
LIN {X 0,Y 177.586,Z 451.383,A -85,B 0,C 180,E1 -22573.017,E2 -22573.017} C_VEL
LIN {X 0,Y 178.624,Z 446.193,A -85,B 0,C 180,E1 -22575.765,E2 -22575.765} C_VEL
LIN {X 0,Y 180.01,Z 440.132,A -85,B 0,C 180,E1 -22578.313,E2 -22578.313} C_VEL
LIN {X 0,Y 181.372,Z 433.644,A -85,B 0,C 180,E1 -22580.521,E2 -22580.521} C_VEL
LIN {X 0,Y 183.126,Z 425.198,A -85,B 0,C 180,E1 -22582.835,E2 -22582.835} C_VEL
LIN {X 0,Y 184.86,Z 415.667,A -85,B 0,C 180,E1 -22584.832,E2 -22584.832} C_VEL
LIN {X 0,Y 186.19,Z 407.246,A -85,B 0,C 180,E1 -22586.213,E2 -22586.213} C_VEL
LIN {X 0,Y 187.224,Z 398.769,A -85,B 0,C 180,E1 -22587.311,E2 -22587.311} C_VEL
LIN {X 0,Y 188.226,Z 389.111,A -85,B 0,C 180,E1 -22588.231,E2 -22588.231} C_VEL
LIN {X 0,Y 188.869,Z 380.199,A -85,B 0,C 180,E1 -22588.817,E2 -22588.817} C_VEL
LIN {X 0,Y 190.475,Z 339.977,A -85,B 0,C 180,E1 -22590.43,E2 -22590.43} C_VEL
LIN {X 0,Y 189.586,Z 335.354,A -85,B 0,C 180,E1 -22590.743,E2 -22590.743} C_VEL
LIN {X 0,Y 184.378,Z 319.805,A -85,B 0,C 180,E1 -22592.128,E2 -22592.128} C_VEL
LIN {X 0,Y 179.196,Z 309.041,A -85,B 0,C 180,E1 -22593.373,E2 -22593.373} C_VEL
LIN {X 0,Y 178.971,Z 308.004,A -85,B 0,C 180,E1 -22593.489,E2 -22593.489} C_VEL
LIN {X 0,Y 178.91,Z 308.012,A -85,B 0,C 180,E1 -22599.04,E2 -22599.04} C_VEL
LIN {X 0,Y 178.653,Z 308.036,A -85,B 0,C 180,E1 -22603.652,E2 -22603.652} C_VEL
LIN {X 0,Y 178.61,Z 308.038,A -85,B 0,C 180,E1 -22609.202,E2 -22609.202} C_VEL
LIN {X 0,Y 178.52,Z 308.056,A -85,B 0,C 180,E1 -22615.113,E2 -22615.113} C_VEL
LIN {X 0,Y 178.501,Z 308.062,A -85,B 0,C 180,E1 -22620.785,E2 -22620.785} C_VEL
LIN {X 0,Y 178.485,Z 308.06,A -85,B 0,C 180,E1 -22624.218,E2 -22624.218} C_VEL
LIN {X 0,Y 178.396,Z 308.075,A -85,B 0,C 180,E1 -22629.073,E2 -22629.073} C_VEL
LIN {X 0,Y 178.413,Z 308.058,A -85,B 0,C 180,E1 -22632.039,E2 -22632.039} C_VEL
LIN {X 0,Y 178.442,Z 308.063,A -85,B 0,C 180,E1 -22635.147,E2 -22635.147} C_VEL
LIN {X 0,Y 178.48,Z 308.064,A -85,B 0,C 180,E1 -22638.429,E2 -22638.429} C_VEL
LIN {X 0,Y 178.457,Z 308.049,A -85,B 0,C 180,E1 -22643.791,E2 -22643.791} C_VEL
LIN {X 0,Y 178.488,Z 308.051,A -85,B 0,C 180,E1 -22646.547,E2 -22646.547} C_VEL
LIN {X 0,Y 178.52,Z 308.058,A -85,B 0,C 180,E1 -22650.005,E2 -22650.005} C_VEL
LIN {X 0,Y 178.521,Z 308.053,A -85,B 0,C 180,E1 -22654.882,E2 -22654.882} C_VEL
LIN {X 0,Y 178.619,Z 308.028,A -85,B 0,C 180,E1 -22660.784,E2 -22660.784} C_VEL
LIN {X 0,Y 178.652,Z 308.043,A -85,B 0,C 180,E1 -22666.347,E2 -22666.347} C_VEL
LIN {X 0,Y 178.906,Z 308.004,A -85,B 0,C 180,E1 -22670.959,E2 -22670.959} C_VEL
LIN {X 0,Y 179.145,Z 307.972,A -85,B 0,C 180,E1 -22677.751,E2 -22677.751} C_VEL
LIN {X 0,Y 179.363,Z 307.95,A -85,B 0,C 180,E1 -22680,E2 -22680} C_VEL
LIN {X 0,Y 178.859,Z 308.015,A -85,B 0,C 180,E1 -22684.507,E2 -22684.507} C_VEL
LIN {X 0,Y 178.906,Z 307.993,A -85,B 0,C 180,E1 -22689.04,E2 -22689.04} C_VEL
LIN {X 0,Y 178.651,Z 308.041,A -85,B 0,C 180,E1 -22693.652,E2 -22693.652} C_VEL
LIN {X 0,Y 178.616,Z 308.043,A -85,B 0,C 180,E1 -22699.214,E2 -22699.214} C_VEL
LIN {X 0,Y 178.515,Z 308.059,A -85,B 0,C 180,E1 -22705.114,E2 -22705.114} C_VEL
LIN {X 0,Y 178.517,Z 308.053,A -85,B 0,C 180,E1 -22709.993,E2 -22709.993} C_VEL
LIN {X 0,Y 178.48,Z 308.068,A -85,B 0,C 180,E1 -22714.219,E2 -22714.219} C_VEL
LIN {X 0,Y 178.391,Z 308.061,A -85,B 0,C 180,E1 -22719.075,E2 -22719.075} C_VEL
LIN {X 0,Y 178.395,Z 308.057,A -85,B 0,C 180,E1 -22722.046,E2 -22722.046} C_VEL
LIN {X 0,Y 178.391,Z 308.076,A -85,B 0,C 180,E1 -22725.164,E2 -22725.164} C_VEL
LIN {X 0,Y 178.401,Z 308.075,A -85,B 0,C 180,E1 -22728.46,E2 -22728.46} C_VEL
LIN {X 0,Y 178.433,Z 308.07,A -85,B 0,C 180,E1 -22733.787,E2 -22733.787} C_VEL
LIN {X 0,Y 178.507,Z 308.176,A -85,B 0,C 180,E1 -22735.423,E2 -22735.423} C_VEL
LIN {X 0,Y 179.566,Z 313.09,A -85,B 0,C 180,E1 -22738.478,E2 -22738.478} C_VEL
LIN {X 0,Y 185.825,Z 330.718,A -85,B 0,C 180,E1 -22740.17,E2 -22740.17} C_VEL
LIN {X 0,Y 186.958,Z 336.463,A -85,B 0,C 180,E1 -22740.575,E2 -22740.575} C_VEL
LIN {X 0,Y 189.858,Z 362.19,A -85,B 0,C 180,E1 -22742.063,E2 -22742.063} C_VEL
LIN {X 0,Y 188.572,Z 391.605,A -85,B 0,C 180,E1 -22743.271,E2 -22743.271} C_VEL
LIN {X 0,Y 187.561,Z 402.609,A -85,B 0,C 180,E1 -22744.051,E2 -22744.051} C_VEL
LIN {X 0,Y 186.227,Z 413.338,A -85,B 0,C 180,E1 -22745.243,E2 -22745.243} C_VEL
LIN {X 0,Y 184.732,Z 423.256,A -85,B 0,C 180,E1 -22746.753,E2 -22746.753} C_VEL
LIN {X 0,Y 183.104,Z 431.375,A -85,B 0,C 180,E1 -22748.32,E2 -22748.32} C_VEL
LIN {X 0,Y 182.148,Z 436.983,A -85,B 0,C 180,E1 -22749.647,E2 -22749.647} C_VEL
LIN {X 0,Y 180.524,Z 441.456,A -85,B 0,C 180,E1 -22750.788,E2 -22750.788} C_VEL
LIN {X 0,Y 176.235,Z 448.082,A -85,B 0,C 180,E1 -22752.774,E2 -22752.774} C_VEL
LIN {X 0,Y 172.127,Z 453.917,A -85,B 0,C 180,E1 -22755.02,E2 -22755.02} C_VEL
LIN {X 0,Y 170.768,Z 457.119,A -85,B 0,C 180,E1 -22756.577,E2 -22756.577} C_VEL
LIN {X 0,Y 169.616,Z 463.477,A -85,B 0,C 180,E1 -22760.46,E2 -22760.46} C_VEL
LIN {X 0,Y 169.176,Z 466.464,A -85,B 0,C 180,E1 -22762.841,E2 -22762.841} C_VEL
LIN {X 0,Y 168.947,Z 468.782,A -85,B 0,C 180,E1 -22765.228,E2 -22765.228} C_VEL
LIN {X 0,Y 168.926,Z 470.484,A -85,B 0,C 180,E1 -22767.616,E2 -22767.616} C_VEL
LIN {X 0,Y 169.012,Z 471.674,A -85,B 0,C 180,E1 -22770,E2 -22770} C_VEL
LIN {X 0,Y 168.873,Z 472.419,A -85,B 0,C 180,E1 -22772.801,E2 -22772.801} C_VEL
LIN {X 0,Y 168.936,Z 472.598,A -85,B 0,C 180,E1 -22774.773,E2 -22774.773} C_VEL
LIN {X 0,Y 169.178,Z 472.242,A -85,B 0,C 180,E1 -22777.159,E2 -22777.159} C_VEL
LIN {X 0,Y 169.65,Z 471.384,A -85,B 0,C 180,E1 -22779.538,E2 -22779.538} C_VEL
LIN {X 0,Y 170.397,Z 470.064,A -85,B 0,C 180,E1 -22781.901,E2 -22781.901} C_VEL
LIN {X 0,Y 172.019,Z 467.096,A -85,B 0,C 180,E1 -22785.4,E2 -22785.4} C_VEL
LIN {X 0,Y 173.456,Z 464.416,A -85,B 0,C 180,E1 -22787.69,E2 -22787.69} C_VEL
LIN {X 0,Y 176.154,Z 459.214,A -85,B 0,C 180,E1 -22791.042,E2 -22791.042} C_VEL
LIN {X 0,Y 179.501,Z 452.405,A -85,B 0,C 180,E1 -22794.273,E2 -22794.273} C_VEL
LIN {X 0,Y 182.762,Z 444.997,A -85,B 0,C 180,E1 -22796.861,E2 -22796.861} C_VEL
LIN {X 0,Y 185.553,Z 437.735,A -85,B 0,C 180,E1 -22798.875,E2 -22798.875} C_VEL
LIN {X 0,Y 188.197,Z 430.404,A -85,B 0,C 180,E1 -22800.476,E2 -22800.476} C_VEL
LIN {X 0,Y 190.274,Z 423.361,A -85,B 0,C 180,E1 -22801.758,E2 -22801.758} C_VEL
LIN {X 0,Y 192.423,Z 415.322,A -85,B 0,C 180,E1 -22802.906,E2 -22802.906} C_VEL
LIN {X 0,Y 194.524,Z 406.064,A -85,B 0,C 180,E1 -22803.899,E2 -22803.899} C_VEL
LIN {X 0,Y 196.274,Z 395.569,A -85,B 0,C 180,E1 -22804.718,E2 -22804.718} C_VEL
LIN {X 0,Y 197.655,Z 381.225,A -85,B 0,C 180,E1 -22805.385,E2 -22805.385} C_VEL
LIN {X 0,Y 198.382,Z 366.499,A -85,B 0,C 180,E1 -22805.974,E2 -22805.974} C_VEL
LIN {X 0,Y 197.261,Z 356.615,A -85,B 0,C 180,E1 -22806.819,E2 -22806.819} C_VEL
LIN {X 0,Y 193.446,Z 347.156,A -85,B 0,C 180,E1 -22808.472,E2 -22808.472} C_VEL
LIN {X 0,Y 188.36,Z 336.583,A -85,B 0,C 180,E1 -22810.768,E2 -22810.768} C_VEL
LIN {X 0,Y 182.866,Z 327.058,A -85,B 0,C 180,E1 -22813.438,E2 -22813.438} C_VEL
LIN {X 0,Y 179.045,Z 321.112,A -85,B 0,C 180,E1 -22815.486,E2 -22815.486} C_VEL
LIN {X 0,Y 176.138,Z 316.509,A -85,B 0,C 180,E1 -22817.201,E2 -22817.201} C_VEL
LIN {X 0,Y 172.266,Z 311.612,A -85,B 0,C 180,E1 -22819.628,E2 -22819.628} C_VEL
LIN {X 0,Y 171.583,Z 310.058,A -85,B 0,C 180,E1 -22820.261,E2 -22820.261} C_VEL
LIN {X 0,Y 171.383,Z 308.941,A -85,B 0,C 180,E1 -22821.717,E2 -22821.717} C_VEL
LIN {X 0,Y 171.394,Z 308.949,A -85,B 0,C 180,E1 -22825.092,E2 -22825.092} C_VEL
LIN {X 0,Y 171.444,Z 308.937,A -85,B 0,C 180,E1 -22830.534,E2 -22830.534} C_VEL
LIN {X 0,Y 171.44,Z 308.94,A -85,B 0,C 180,E1 -22835.799,E2 -22835.799} C_VEL
LIN {X 0,Y 171.572,Z 308.924,A -85,B 0,C 180,E1 -22840.871,E2 -22840.871} C_VEL
LIN {X 0,Y 171.569,Z 308.91,A -85,B 0,C 180,E1 -22845.772,E2 -22845.772} C_VEL
LIN {X 0,Y 171.845,Z 308.868,A -85,B 0,C 180,E1 -22850.585,E2 -22850.585} C_VEL
LIN {X 0,Y 171.807,Z 308.879,A -85,B 0,C 180,E1 -22855.308,E2 -22855.308} C_VEL
LIN {X 0,Y 172.325,Z 308.828,A -85,B 0,C 180,E1 -22860,E2 -22860} C_VEL
LIN {X 0,Y 171.799,Z 308.895,A -85,B 0,C 180,E1 -22864.693,E2 -22864.693} C_VEL
LIN {X 0,Y 171.836,Z 308.886,A -85,B 0,C 180,E1 -22869.416,E2 -22869.416} C_VEL
LIN {X 0,Y 171.655,Z 308.903,A -85,B 0,C 180,E1 -22872.215,E2 -22872.215} C_VEL
LIN {X 0,Y 172.394,Z 311.37,A -85,B 0,C 180,E1 -22872.884,E2 -22872.884} C_VEL
LIN {X 0,Y 174.371,Z 313.694,A -85,B 0,C 180,E1 -22874.144,E2 -22874.144} C_VEL
LIN {X 0,Y 175.722,Z 314.797,A -85,B 0,C 180,E1 -22874.92,E2 -22874.92} C_VEL
LIN {X 0,Y 177.505,Z 317.82,A -85,B 0,C 180,E1 -22876.017,E2 -22876.017} C_VEL
LIN {X 0,Y 179.484,Z 319.911,A -85,B 0,C 180,E1 -22877.078,E2 -22877.078} C_VEL
LIN {X 0,Y 182.063,Z 323.595,A -85,B 0,C 180,E1 -22878.457,E2 -22878.457} C_VEL
LIN {X 0,Y 186.464,Z 330.009,A -85,B 0,C 180,E1 -22880.591,E2 -22880.591} C_VEL
LIN {X 0,Y 190.579,Z 336.44,A -85,B 0,C 180,E1 -22882.44,E2 -22882.44} C_VEL
LIN {X 0,Y 194.746,Z 343.852,A -85,B 0,C 180,E1 -22884.192,E2 -22884.192} C_VEL
LIN {X 0,Y 199.077,Z 353.821,A -85,B 0,C 180,E1 -22885.992,E2 -22885.992} C_VEL
LIN {X 0,Y 197.232,Z 382.382,A -85,B 0,C 180,E1 -22887.115,E2 -22887.115} C_VEL
LIN {X 0,Y 195.765,Z 394.046,A -85,B 0,C 180,E1 -22887.879,E2 -22887.879} C_VEL
LIN {X 0,Y 193.719,Z 404.958,A -85,B 0,C 180,E1 -22889.021,E2 -22889.021} C_VEL
LIN {X 0,Y 191.47,Z 414.153,A -85,B 0,C 180,E1 -22890.311,E2 -22890.311} C_VEL
LIN {X 0,Y 189.072,Z 422.254,A -85,B 0,C 180,E1 -22891.76,E2 -22891.76} C_VEL
LIN {X 0,Y 186.477,Z 429.96,A -85,B 0,C 180,E1 -22893.506,E2 -22893.506} C_VEL
LIN {X 0,Y 183.414,Z 437.758,A -85,B 0,C 180,E1 -22895.72,E2 -22895.72} C_VEL
LIN {X 0,Y 179.802,Z 445.682,A -85,B 0,C 180,E1 -22898.712,E2 -22898.712} C_VEL
LIN {X 0,Y 177.336,Z 450.623,A -85,B 0,C 180,E1 -22901.152,E2 -22901.152} C_VEL
LIN {X 0,Y 175.169,Z 454.759,A -85,B 0,C 180,E1 -22903.767,E2 -22903.767} C_VEL
LIN {X 0,Y 172.867,Z 458.61,A -85,B 0,C 180,E1 -22907.038,E2 -22907.038} C_VEL
LIN {X 0,Y 171.744,Z 460.424,A -85,B 0,C 180,E1 -22909.102,E2 -22909.102} C_VEL
LIN {X 0,Y 170.49,Z 462.128,A -85,B 0,C 180,E1 -22911.807,E2 -22911.807} C_VEL
LIN {X 0,Y 169.604,Z 463.145,A -85,B 0,C 180,E1 -22914.542,E2 -22914.542} C_VEL
LIN {X 0,Y 168.998,Z 463.472,A -85,B 0,C 180,E1 -22917.275,E2 -22917.275} C_VEL
LIN {X 0,Y 168.6,Z 462.805,A -85,B 0,C 180,E1 -22921.09,E2 -22921.09} C_VEL
LIN {X 0,Y 168.734,Z 460.505,A -85,B 0,C 180,E1 -22925.386,E2 -22925.386} C_VEL
LIN {X 0,Y 169.455,Z 456.905,A -85,B 0,C 180,E1 -22929.359,E2 -22929.359} C_VEL
LIN {X 0,Y 170.3,Z 452.661,A -85,B 0,C 180,E1 -22932.557,E2 -22932.557} C_VEL
LIN {X 0,Y 171.471,Z 447.016,A -85,B 0,C 180,E1 -22935.764,E2 -22935.764} C_VEL
LIN {X 0,Y 172.736,Z 441.479,A -85,B 0,C 180,E1 -22938.263,E2 -22938.263} C_VEL
LIN {X 0,Y 174.244,Z 434.744,A -85,B 0,C 180,E1 -22940.716,E2 -22940.716} C_VEL
LIN {X 0,Y 176.023,Z 426.487,A -85,B 0,C 180,E1 -22943.121,E2 -22943.121} C_VEL
LIN {X 0,Y 178.087,Z 415.883,A -85,B 0,C 180,E1 -22945.473,E2 -22945.473} C_VEL
LIN {X 0,Y 179.469,Z 407.39,A -85,B 0,C 180,E1 -22946.914,E2 -22946.914} C_VEL
LIN {X 0,Y 180.558,Z 398.889,A -85,B 0,C 180,E1 -22948.048,E2 -22948.048} C_VEL
LIN {X 0,Y 181.557,Z 389.672,A -85,B 0,C 180,E1 -22948.96,E2 -22948.96} C_VEL
LIN {X 0,Y 182.235,Z 380.603,A -85,B 0,C 180,E1 -22949.586,E2 -22949.586} C_VEL
LIN {X 0,Y 183.959,Z 341.173,A -85,B 0,C 180,E1 -22951.213,E2 -22951.213} C_VEL
LIN {X 0,Y 183.035,Z 336.86,A -85,B 0,C 180,E1 -22951.534,E2 -22951.534} C_VEL
LIN {X 0,Y 178.26,Z 322.557,A -85,B 0,C 180,E1 -22952.877,E2 -22952.877} C_VEL
LIN {X 0,Y 172.843,Z 311.699,A -85,B 0,C 180,E1 -22954.235,E2 -22954.235} C_VEL
LIN {X 0,Y 171.832,Z 308.891,A -85,B 0,C 180,E1 -22954.545,E2 -22954.545} C_VEL
LIN {X 0,Y 171.848,Z 308.892,A -85,B 0,C 180,E1 -22959.415,E2 -22959.415} C_VEL
LIN {X 0,Y 171.57,Z 308.92,A -85,B 0,C 180,E1 -22964.227,E2 -22964.227} C_VEL
LIN {X 0,Y 171.531,Z 308.916,A -85,B 0,C 180,E1 -22969.548,E2 -22969.548} C_VEL
LIN {X 0,Y 171.46,Z 308.939,A -85,B 0,C 180,E1 -22975.608,E2 -22975.608} C_VEL
LIN {X 0,Y 171.459,Z 308.94,A -85,B 0,C 180,E1 -22980.595,E2 -22980.595} C_VEL
LIN {X 0,Y 171.392,Z 308.946,A -85,B 0,C 180,E1 -22985.034,E2 -22985.034} C_VEL
LIN {X 0,Y 171.358,Z 308.953,A -85,B 0,C 180,E1 -22988.807,E2 -22988.807} C_VEL
LIN {X 0,Y 171.354,Z 308.945,A -85,B 0,C 180,E1 -22994.205,E2 -22994.205} C_VEL
LIN {X 0,Y 171.403,Z 308.946,A -85,B 0,C 180,E1 -22999.001,E2 -22999.001} C_VEL
LIN {X 0,Y 171.435,Z 308.933,A -85,B 0,C 180,E1 -23002.053,E2 -23002.053} C_VEL
LIN {X 0,Y 171.417,Z 308.935,A -85,B 0,C 180,E1 -23007.792,E2 -23007.792} C_VEL
LIN {X 0,Y 171.446,Z 308.94,A -85,B 0,C 180,E1 -23010.534,E2 -23010.534} C_VEL
LIN {X 0,Y 171.449,Z 308.932,A -85,B 0,C 180,E1 -23015.8,E2 -23015.8} C_VEL
LIN {X 0,Y 171.575,Z 308.905,A -85,B 0,C 180,E1 -23020.871,E2 -23020.871} C_VEL
LIN {X 0,Y 171.57,Z 308.923,A -85,B 0,C 180,E1 -23025.772,E2 -23025.772} C_VEL
LIN {X 0,Y 171.843,Z 308.886,A -85,B 0,C 180,E1 -23030.584,E2 -23030.584} C_VEL
LIN {X 0,Y 171.806,Z 308.871,A -85,B 0,C 180,E1 -23035.307,E2 -23035.307} C_VEL
LIN {X 0,Y 172.326,Z 308.827,A -85,B 0,C 180,E1 -23040,E2 -23040} C_VEL
LIN {X 0,Y 171.807,Z 308.894,A -85,B 0,C 180,E1 -23044.692,E2 -23044.692} C_VEL
LIN {X 0,Y 171.843,Z 308.872,A -85,B 0,C 180,E1 -23049.415,E2 -23049.415} C_VEL
LIN {X 0,Y 171.569,Z 308.924,A -85,B 0,C 180,E1 -23054.228,E2 -23054.228} C_VEL
LIN {X 0,Y 171.535,Z 308.921,A -85,B 0,C 180,E1 -23059.557,E2 -23059.557} C_VEL
LIN {X 0,Y 171.454,Z 308.94,A -85,B 0,C 180,E1 -23065.609,E2 -23065.609} C_VEL
LIN {X 0,Y 171.436,Z 308.934,A -85,B 0,C 180,E1 -23070.586,E2 -23070.586} C_VEL
LIN {X 0,Y 171.389,Z 308.949,A -85,B 0,C 180,E1 -23075.035,E2 -23075.035} C_VEL
LIN {X 0,Y 171.354,Z 308.938,A -85,B 0,C 180,E1 -23078.808,E2 -23078.808} C_VEL
LIN {X 0,Y 171.318,Z 308.952,A -85,B 0,C 180,E1 -23084.218,E2 -23084.218} C_VEL
LIN {X 0,Y 171.333,Z 308.957,A -85,B 0,C 180,E1 -23088.982,E2 -23088.982} C_VEL
LIN {X 0,Y 171.41,Z 308.946,A -85,B 0,C 180,E1 -23094.25,E2 -23094.25} C_VEL
LIN {X 0,Y 171.437,Z 308.963,A -85,B 0,C 180,E1 -23094.797,E2 -23094.797} C_VEL
LIN {X 0,Y 172.277,Z 312.819,A -85,B 0,C 180,E1 -23097.329,E2 -23097.329} C_VEL
LIN {X 0,Y 178.698,Z 330.494,A -85,B 0,C 180,E1 -23099.171,E2 -23099.171} C_VEL
LIN {X 0,Y 180.22,Z 335.732,A -85,B 0,C 180,E1 -23099.633,E2 -23099.633} C_VEL
LIN {X 0,Y 183.248,Z 362.858,A -85,B 0,C 180,E1 -23101.281,E2 -23101.281} C_VEL
LIN {X 0,Y 182.001,Z 390.761,A -85,B 0,C 180,E1 -23102.462,E2 -23102.462} C_VEL
LIN {X 0,Y 181.081,Z 400.939,A -85,B 0,C 180,E1 -23103.182,E2 -23103.182} C_VEL
LIN {X 0,Y 179.724,Z 411.854,A -85,B 0,C 180,E1 -23104.348,E2 -23104.348} C_VEL
LIN {X 0,Y 178.243,Z 421.723,A -85,B 0,C 180,E1 -23105.854,E2 -23105.854} C_VEL
LIN {X 0,Y 176.512,Z 430.076,A -85,B 0,C 180,E1 -23107.467,E2 -23107.467} C_VEL
LIN {X 0,Y 175.23,Z 437.014,A -85,B 0,C 180,E1 -23109.149,E2 -23109.149} C_VEL
LIN {X 0,Y 173.743,Z 443.742,A -85,B 0,C 180,E1 -23111.12,E2 -23111.12} C_VEL
LIN {X 0,Y 172.254,Z 450.117,A -85,B 0,C 180,E1 -23113.406,E2 -23113.406} C_VEL
LIN {X 0,Y 171.132,Z 455.418,A -85,B 0,C 180,E1 -23115.735,E2 -23115.735} C_VEL
LIN {X 0,Y 170.768,Z 457.119,A -85,B 0,C 180,E1 -23116.577,E2 -23116.577} C_VEL
LIN {X 0,Y 169.496,Z 460.196,A -85,B 0,C 180,E1 -23118.223,E2 -23118.223} C_VEL
LIN {X 0,Y 167.427,Z 462.825,A -85,B 0,C 180,E1 -23119.898,E2 -23119.898} C_VEL
LIN {X 0,Y 163.092,Z 466.971,A -85,B 0,C 180,E1 -23123.491,E2 -23123.491} C_VEL
LIN {X 0,Y 161.844,Z 468.992,A -85,B 0,C 180,E1 -23125.803,E2 -23125.803} C_VEL
LIN {X 0,Y 161.816,Z 469.139,A -85,B 0,C 180,E1 -23126.143,E2 -23126.143} C_VEL
LIN {X 0,Y 161.922,Z 471.37,A -85,B 0,C 180,E1 -23130,E2 -23130} C_VEL
LIN {X 0,Y 161.796,Z 472.136,A -85,B 0,C 180,E1 -23132.489,E2 -23132.489} C_VEL
LIN {X 0,Y 161.857,Z 472.4,A -85,B 0,C 180,E1 -23134.982,E2 -23134.982} C_VEL
LIN {X 0,Y 162.139,Z 472.082,A -85,B 0,C 180,E1 -23137.471,E2 -23137.471} C_VEL
LIN {X 0,Y 162.635,Z 471.302,A -85,B 0,C 180,E1 -23139.953,E2 -23139.953} C_VEL
LIN {X 0,Y 163.454,Z 470.064,A -85,B 0,C 180,E1 -23142.414,E2 -23142.414} C_VEL
LIN {X 0,Y 165.178,Z 467.179,A -85,B 0,C 180,E1 -23146.055,E2 -23146.055} C_VEL
LIN {X 0,Y 167.537,Z 463.057,A -85,B 0,C 180,E1 -23149.608,E2 -23149.608} C_VEL
LIN {X 0,Y 170.655,Z 457.519,A -85,B 0,C 180,E1 -23153.03,E2 -23153.03} C_VEL
LIN {X 0,Y 173.679,Z 451.487,A -85,B 0,C 180,E1 -23155.785,E2 -23155.785} C_VEL
LIN {X 0,Y 176.496,Z 445.624,A -85,B 0,C 180,E1 -23157.896,E2 -23157.896} C_VEL
LIN {X 0,Y 179.411,Z 438.55,A -85,B 0,C 180,E1 -23159.963,E2 -23159.963} C_VEL
LIN {X 0,Y 182.613,Z 430.079,A -85,B 0,C 180,E1 -23161.878,E2 -23161.878} C_VEL
LIN {X 0,Y 184.775,Z 423.22,A -85,B 0,C 180,E1 -23163.143,E2 -23163.143} C_VEL
LIN {X 0,Y 187.049,Z 415.207,A -85,B 0,C 180,E1 -23164.303,E2 -23164.303} C_VEL
LIN {X 0,Y 189.231,Z 406.011,A -85,B 0,C 180,E1 -23165.308,E2 -23165.308} C_VEL
LIN {X 0,Y 190.928,Z 396.377,A -85,B 0,C 180,E1 -23166.081,E2 -23166.081} C_VEL
LIN {X 0,Y 192.232,Z 385.102,A -85,B 0,C 180,E1 -23166.675,E2 -23166.675} C_VEL
LIN {X 0,Y 193.202,Z 367.574,A -85,B 0,C 180,E1 -23167.382,E2 -23167.382} C_VEL
LIN {X 0,Y 192.322,Z 359.452,A -85,B 0,C 180,E1 -23168.107,E2 -23168.107} C_VEL
LIN {X 0,Y 188.651,Z 350.32,A -85,B 0,C 180,E1 -23169.815,E2 -23169.815} C_VEL
LIN {X 0,Y 184.295,Z 341.065,A -85,B 0,C 180,E1 -23171.948,E2 -23171.948} C_VEL
LIN {X 0,Y 179.443,Z 332.341,A -85,B 0,C 180,E1 -23174.482,E2 -23174.482} C_VEL
LIN {X 0,Y 175.798,Z 326.547,A -85,B 0,C 180,E1 -23176.573,E2 -23176.573} C_VEL
LIN {X 0,Y 172.724,Z 321.727,A -85,B 0,C 180,E1 -23178.501,E2 -23178.501} C_VEL
LIN {X 0,Y 169.171,Z 316.621,A -85,B 0,C 180,E1 -23180.976,E2 -23180.976} C_VEL
LIN {X 0,Y 167.739,Z 315.033,A -85,B 0,C 180,E1 -23182.021,E2 -23182.021} C_VEL
LIN {X 0,Y 165.449,Z 312.905,A -85,B 0,C 180,E1 -23183.81,E2 -23183.81} C_VEL
LIN {X 0,Y 164.46,Z 310.541,A -85,B 0,C 180,E1 -23184.807,E2 -23184.807} C_VEL
LIN {X 0,Y 164.347,Z 309.827,A -85,B 0,C 180,E1 -23184.988,E2 -23184.988} C_VEL
LIN {X 0,Y 164.385,Z 309.813,A -85,B 0,C 180,E1 -23189.134,E2 -23189.134} C_VEL
LIN {X 0,Y 164.402,Z 309.812,A -85,B 0,C 180,E1 -23194.692,E2 -23194.692} C_VEL
LIN {X 0,Y 164.48,Z 309.797,A -85,B 0,C 180,E1 -23200.051,E2 -23200.051} C_VEL
LIN {X 0,Y 164.499,Z 309.786,A -85,B 0,C 180,E1 -23205.147,E2 -23205.147} C_VEL
LIN {X 0,Y 164.764,Z 309.751,A -85,B 0,C 180,E1 -23210.176,E2 -23210.176} C_VEL
LIN {X 0,Y 164.827,Z 309.754,A -85,B 0,C 180,E1 -23212.651,E2 -23212.651} C_VEL
LIN {X 0,Y 165.04,Z 309.718,A -85,B 0,C 180,E1 -23217.56,E2 -23217.56} C_VEL
LIN {X 0,Y 165.288,Z 309.704,A -85,B 0,C 180,E1 -23220,E2 -23220} C_VEL
LIN {X 0,Y 164.748,Z 309.774,A -85,B 0,C 180,E1 -23224.895,E2 -23224.895} C_VEL
LIN {X 0,Y 164.783,Z 309.767,A -85,B 0,C 180,E1 -23227.814,E2 -23227.814} C_VEL
LIN {X 0,Y 165.525,Z 312.129,A -85,B 0,C 180,E1 -23228.623,E2 -23228.623} C_VEL
LIN {X 0,Y 167.486,Z 314.54,A -85,B 0,C 180,E1 -23230.228,E2 -23230.228} C_VEL
LIN {X 0,Y 169.042,Z 315.699,A -85,B 0,C 180,E1 -23231.315,E2 -23231.315} C_VEL
LIN {X 0,Y 170.783,Z 318.797,A -85,B 0,C 180,E1 -23232.628,E2 -23232.628} C_VEL
LIN {X 0,Y 173.012,Z 321.072,A -85,B 0,C 180,E1 -23234.059,E2 -23234.059} C_VEL
LIN {X 0,Y 175.291,Z 324.429,A -85,B 0,C 180,E1 -23235.478,E2 -23235.478} C_VEL
LIN {X 0,Y 176.643,Z 326.021,A -85,B 0,C 180,E1 -23236.246,E2 -23236.246} C_VEL
LIN {X 0,Y 182.543,Z 334.614,A -85,B 0,C 180,E1 -23239.413,E2 -23239.413} C_VEL
LIN {X 0,Y 187.601,Z 342.829,A -85,B 0,C 180,E1 -23241.815,E2 -23241.815} C_VEL
LIN {X 0,Y 190.93,Z 349.23,A -85,B 0,C 180,E1 -23243.328,E2 -23243.328} C_VEL
LIN {X 0,Y 193.925,Z 356.24,A -85,B 0,C 180,E1 -23244.65,E2 -23244.65} C_VEL
LIN {X 0,Y 192.056,Z 382.649,A -85,B 0,C 180,E1 -23245.691,E2 -23245.691} C_VEL
LIN {X 0,Y 190.562,Z 394.116,A -85,B 0,C 180,E1 -23246.452,E2 -23246.452} C_VEL
LIN {X 0,Y 188.387,Z 405.201,A -85,B 0,C 180,E1 -23247.626,E2 -23247.626} C_VEL
LIN {X 0,Y 186.363,Z 413.225,A -85,B 0,C 180,E1 -23248.746,E2 -23248.746} C_VEL
LIN {X 0,Y 183.886,Z 421.25,A -85,B 0,C 180,E1 -23250.154,E2 -23250.154} C_VEL
LIN {X 0,Y 181.572,Z 427.949,A -85,B 0,C 180,E1 -23251.623,E2 -23251.623} C_VEL
LIN {X 0,Y 178.764,Z 435.027,A -85,B 0,C 180,E1 -23253.542,E2 -23253.542} C_VEL
LIN {X 0,Y 176.421,Z 440.259,A -85,B 0,C 180,E1 -23255.252,E2 -23255.252} C_VEL
LIN {X 0,Y 172.888,Z 447.279,A -85,B 0,C 180,E1 -23258.18,E2 -23258.18} C_VEL
LIN {X 0,Y 170.694,Z 451.391,A -85,B 0,C 180,E1 -23260.371,E2 -23260.371} C_VEL
LIN {X 0,Y 168.412,Z 455.426,A -85,B 0,C 180,E1 -23263.091,E2 -23263.091} C_VEL
LIN {X 0,Y 166.329,Z 458.628,A -85,B 0,C 180,E1 -23265.916,E2 -23265.916} C_VEL
LIN {X 0,Y 165.556,Z 459.856,A -85,B 0,C 180,E1 -23267.219,E2 -23267.219} C_VEL
LIN {X 0,Y 163.912,Z 462.081,A -85,B 0,C 180,E1 -23270.514,E2 -23270.514} C_VEL
LIN {X 0,Y 162.979,Z 463.009,A -85,B 0,C 180,E1 -23272.865,E2 -23272.865} C_VEL
LIN {X 0,Y 162.19,Z 463.564,A -85,B 0,C 180,E1 -23275.716,E2 -23275.716} C_VEL
LIN {X 0,Y 161.544,Z 463.118,A -85,B 0,C 180,E1 -23280.472,E2 -23280.472} C_VEL
LIN {X 0,Y 161.528,Z 461.394,A -85,B 0,C 180,E1 -23284.21,E2 -23284.21} C_VEL
LIN {X 0,Y 161.88,Z 459.388,A -85,B 0,C 180,E1 -23287.001,E2 -23287.001} C_VEL
LIN {X 0,Y 162.697,Z 455.375,A -85,B 0,C 180,E1 -23290.819,E2 -23290.819} C_VEL
LIN {X 0,Y 163.58,Z 451.207,A -85,B 0,C 180,E1 -23293.784,E2 -23293.784} C_VEL
LIN {X 0,Y 164.599,Z 446.556,A -85,B 0,C 180,E1 -23296.418,E2 -23296.418} C_VEL
LIN {X 0,Y 165.941,Z 440.887,A -85,B 0,C 180,E1 -23299.013,E2 -23299.013} C_VEL
LIN {X 0,Y 167.538,Z 433.999,A -85,B 0,C 180,E1 -23301.558,E2 -23301.558} C_VEL
LIN {X 0,Y 169.545,Z 425.01,A -85,B 0,C 180,E1 -23304.185,E2 -23304.185} C_VEL
LIN {X 0,Y 171.349,Z 416.029,A -85,B 0,C 180,E1 -23306.179,E2 -23306.179} C_VEL
LIN {X 0,Y 172.786,Z 407.525,A -85,B 0,C 180,E1 -23307.669,E2 -23307.669} C_VEL
LIN {X 0,Y 173.898,Z 399.034,A -85,B 0,C 180,E1 -23308.842,E2 -23308.842} C_VEL
LIN {X 0,Y 174.948,Z 389.79,A -85,B 0,C 180,E1 -23309.784,E2 -23309.784} C_VEL
LIN {X 0,Y 175.669,Z 380.568,A -85,B 0,C 180,E1 -23310.436,E2 -23310.436} C_VEL
LIN {X 0,Y 177.442,Z 342.016,A -85,B 0,C 180,E1 -23312.076,E2 -23312.076} C_VEL
LIN {X 0,Y 175.877,Z 336.499,A -85,B 0,C 180,E1 -23312.567,E2 -23312.567} C_VEL
LIN {X 0,Y 172.256,Z 325.536,A -85,B 0,C 180,E1 -23313.643,E2 -23313.643} C_VEL
LIN {X 0,Y 164.913,Z 310.575,A -85,B 0,C 180,E1 -23315.613,E2 -23315.613} C_VEL
LIN {X 0,Y 164.758,Z 309.766,A -85,B 0,C 180,E1 -23315.814,E2 -23315.814} C_VEL
LIN {X 0,Y 164.768,Z 309.772,A -85,B 0,C 180,E1 -23319.823,E2 -23319.823} C_VEL
LIN {X 0,Y 164.5,Z 309.804,A -85,B 0,C 180,E1 -23324.853,E2 -23324.853} C_VEL
LIN {X 0,Y 164.473,Z 309.788,A -85,B 0,C 180,E1 -23329.989,E2 -23329.989} C_VEL
LIN {X 0,Y 164.387,Z 309.82,A -85,B 0,C 180,E1 -23336.128,E2 -23336.128} C_VEL
LIN {X 0,Y 164.389,Z 309.816,A -85,B 0,C 180,E1 -23341.235,E2 -23341.235} C_VEL
LIN {X 0,Y 164.294,Z 309.833,A -85,B 0,C 180,E1 -23346.788,E2 -23346.788} C_VEL
LIN {X 0,Y 164.292,Z 309.827,A -85,B 0,C 180,E1 -23349.914,E2 -23349.914} C_VEL
LIN {X 0,Y 164.306,Z 309.816,A -85,B 0,C 180,E1 -23353.351,E2 -23353.351} C_VEL
LIN {X 0,Y 164.322,Z 309.826,A -85,B 0,C 180,E1 -23356.818,E2 -23356.818} C_VEL
LIN {X 0,Y 164.366,Z 309.819,A -85,B 0,C 180,E1 -23360.32,E2 -23360.32} C_VEL
LIN {X 0,Y 164.342,Z 309.803,A -85,B 0,C 180,E1 -23364.341,E2 -23364.341} C_VEL
LIN {X 0,Y 164.388,Z 309.815,A -85,B 0,C 180,E1 -23369.134,E2 -23369.134} C_VEL
LIN {X 0,Y 164.407,Z 309.811,A -85,B 0,C 180,E1 -23374.692,E2 -23374.692} C_VEL
LIN {X 0,Y 164.481,Z 309.781,A -85,B 0,C 180,E1 -23380.05,E2 -23380.05} C_VEL
LIN {X 0,Y 164.518,Z 309.802,A -85,B 0,C 180,E1 -23385.148,E2 -23385.148} C_VEL
LIN {X 0,Y 164.763,Z 309.77,A -85,B 0,C 180,E1 -23390.176,E2 -23390.176} C_VEL
LIN {X 0,Y 164.825,Z 309.749,A -85,B 0,C 180,E1 -23392.65,E2 -23392.65} C_VEL
LIN {X 0,Y 165.04,Z 309.724,A -85,B 0,C 180,E1 -23397.559,E2 -23397.559} C_VEL
LIN {X 0,Y 165.289,Z 309.704,A -85,B 0,C 180,E1 -23400,E2 -23400} C_VEL
LIN {X 0,Y 164.756,Z 309.772,A -85,B 0,C 180,E1 -23404.894,E2 -23404.894} C_VEL
LIN {X 0,Y 164.825,Z 309.751,A -85,B 0,C 180,E1 -23407.349,E2 -23407.349} C_VEL
LIN {X 0,Y 164.698,Z 309.766,A -85,B 0,C 180,E1 -23411.06,E2 -23411.06} C_VEL
LIN {X 0,Y 164.477,Z 309.809,A -85,B 0,C 180,E1 -23417.404,E2 -23417.404} C_VEL
LIN {X 0,Y 164.469,Z 309.798,A -85,B 0,C 180,E1 -23419.989,E2 -23419.989} C_VEL
LIN {X 0,Y 164.381,Z 309.823,A -85,B 0,C 180,E1 -23426.128,E2 -23426.128} C_VEL
LIN {X 0,Y 164.37,Z 309.816,A -85,B 0,C 180,E1 -23431.227,E2 -23431.227} C_VEL
LIN {X 0,Y 164.291,Z 309.829,A -85,B 0,C 180,E1 -23436.79,E2 -23436.79} C_VEL
LIN {X 0,Y 164.287,Z 309.81,A -85,B 0,C 180,E1 -23439.917,E2 -23439.917} C_VEL
LIN {X 0,Y 164.277,Z 309.823,A -85,B 0,C 180,E1 -23443.343,E2 -23443.343} C_VEL
LIN {X 0,Y 164.261,Z 309.836,A -85,B 0,C 180,E1 -23446.8,E2 -23446.8} C_VEL
LIN {X 0,Y 164.293,Z 309.832,A -85,B 0,C 180,E1 -23450.353,E2 -23450.353} C_VEL
LIN {X 0,Y 164.41,Z 309.996,A -85,B 0,C 180,E1 -23454.31,E2 -23454.31} C_VEL
LIN {X 0,Y 164.984,Z 312.667,A -85,B 0,C 180,E1 -23456.123,E2 -23456.123} C_VEL
LIN {X 0,Y 172.011,Z 331.349,A -85,B 0,C 180,E1 -23458.211,E2 -23458.211} C_VEL
LIN {X 0,Y 173.914,Z 337.764,A -85,B 0,C 180,E1 -23458.81,E2 -23458.81} C_VEL
LIN {X 0,Y 176.694,Z 363.289,A -85,B 0,C 180,E1 -23460.432,E2 -23460.432} C_VEL
LIN {X 0,Y 175.414,Z 390.596,A -85,B 0,C 180,E1 -23461.629,E2 -23461.629} C_VEL
LIN {X 0,Y 174.492,Z 400.569,A -85,B 0,C 180,E1 -23462.356,E2 -23462.356} C_VEL
LIN {X 0,Y 173.087,Z 410.965,A -85,B 0,C 180,E1 -23463.472,E2 -23463.472} C_VEL
LIN {X 0,Y 171.482,Z 421.684,A -85,B 0,C 180,E1 -23465.161,E2 -23465.161} C_VEL
LIN {X 0,Y 169.685,Z 430.008,A -85,B 0,C 180,E1 -23466.83,E2 -23466.83} C_VEL
LIN {X 0,Y 168.354,Z 436.926,A -85,B 0,C 180,E1 -23468.576,E2 -23468.576} C_VEL
LIN {X 0,Y 166.991,Z 442.773,A -85,B 0,C 180,E1 -23470.325,E2 -23470.325} C_VEL
LIN {X 0,Y 165.442,Z 449.282,A -85,B 0,C 180,E1 -23472.701,E2 -23472.701} C_VEL
LIN {X 0,Y 164.257,Z 454.695,A -85,B 0,C 180,E1 -23475.125,E2 -23475.125} C_VEL
LIN {X 0,Y 163.259,Z 459.195,A -85,B 0,C 180,E1 -23477.571,E2 -23477.571} C_VEL
LIN {X 0,Y 162.598,Z 462.939,A -85,B 0,C 180,E1 -23480.044,E2 -23480.044} C_VEL
LIN {X 0,Y 162.137,Z 465.979,A -85,B 0,C 180,E1 -23482.528,E2 -23482.528} C_VEL
LIN {X 0,Y 161.816,Z 469.139,A -85,B 0,C 180,E1 -23486.143,E2 -23486.143} C_VEL
LIN {X 0,Y 161.472,Z 470.081,A -85,B 0,C 180,E1 -23487.495,E2 -23487.495} C_VEL
LIN {X 0,Y 160.075,Z 471.161,A -85,B 0,C 180,E1 -23489.515,E2 -23489.515} C_VEL
LIN {X 0,Y 156.898,Z 472.016,A -85,B 0,C 180,E1 -23492.926,E2 -23492.926} C_VEL
LIN {X 0,Y 155.03,Z 472.164,A -85,B 0,C 180,E1 -23496.167,E2 -23496.167} C_VEL
LIN {X 0,Y 154.993,Z 471.975,A -85,B 0,C 180,E1 -23497.274,E2 -23497.274} C_VEL
LIN {X 0,Y 155.643,Z 471.222,A -85,B 0,C 180,E1 -23500.405,E2 -23500.405} C_VEL
LIN {X 0,Y 156.532,Z 470.064,A -85,B 0,C 180,E1 -23502.972,E2 -23502.972} C_VEL
LIN {X 0,Y 158.364,Z 467.262,A -85,B 0,C 180,E1 -23506.765,E2 -23506.765} C_VEL
LIN {X 0,Y 160.863,Z 463.238,A -85,B 0,C 180,E1 -23510.457,E2 -23510.457} C_VEL
LIN {X 0,Y 163.013,Z 459.768,A -85,B 0,C 180,E1 -23512.83,E2 -23512.83} C_VEL
LIN {X 0,Y 166.083,Z 454.428,A -85,B 0,C 180,E1 -23515.704,E2 -23515.704} C_VEL
LIN {X 0,Y 168.801,Z 449.207,A -85,B 0,C 180,E1 -23517.929,E2 -23517.929} C_VEL
LIN {X 0,Y 171.845,Z 442.946,A -85,B 0,C 180,E1 -23520.064,E2 -23520.064} C_VEL
LIN {X 0,Y 174.931,Z 435.604,A -85,B 0,C 180,E1 -23522.087,E2 -23522.087} C_VEL
LIN {X 0,Y 178.543,Z 425.836,A -85,B 0,C 180,E1 -23524.166,E2 -23524.166} C_VEL
LIN {X 0,Y 181.287,Z 416.966,A -85,B 0,C 180,E1 -23525.555,E2 -23525.555} C_VEL
LIN {X 0,Y 183.797,Z 407.144,A -85,B 0,C 180,E1 -23526.687,E2 -23526.687} C_VEL
LIN {X 0,Y 185.586,Z 397.828,A -85,B 0,C 180,E1 -23527.481,E2 -23527.481} C_VEL
LIN {X 0,Y 186.784,Z 388.799,A -85,B 0,C 180,E1 -23528.02,E2 -23528.02} C_VEL
LIN {X 0,Y 188.213,Z 369.279,A -85,B 0,C 180,E1 -23528.81,E2 -23528.81} C_VEL
LIN {X 0,Y 187.545,Z 362.412,A -85,B 0,C 180,E1 -23529.445,E2 -23529.445} C_VEL
LIN {X 0,Y 183.442,Z 352.147,A -85,B 0,C 180,E1 -23531.536,E2 -23531.536} C_VEL
LIN {X 0,Y 179.241,Z 343.481,A -85,B 0,C 180,E1 -23533.762,E2 -23533.762} C_VEL
LIN {X 0,Y 175.535,Z 336.792,A -85,B 0,C 180,E1 -23535.899,E2 -23535.899} C_VEL
LIN {X 0,Y 172.644,Z 331.957,A -85,B 0,C 180,E1 -23537.686,E2 -23537.686} C_VEL
LIN {X 0,Y 169.9,Z 327.514,A -85,B 0,C 180,E1 -23539.552,E2 -23539.552} C_VEL
LIN {X 0,Y 166.027,Z 321.802,A -85,B 0,C 180,E1 -23542.464,E2 -23542.464} C_VEL
LIN {X 0,Y 163.486,Z 319.445,A -85,B 0,C 180,E1 -23544.521,E2 -23544.521} C_VEL
LIN {X 0,Y 161.996,Z 316.513,A -85,B 0,C 180,E1 -23546.044,E2 -23546.044} C_VEL
LIN {X 0,Y 159.492,Z 314.994,A -85,B 0,C 180,E1 -23548.445,E2 -23548.445} C_VEL
LIN {X 0,Y 157.693,Z 312.372,A -85,B 0,C 180,E1 -23550.735,E2 -23550.735} C_VEL
LIN {X 0,Y 157.274,Z 310.691,A -85,B 0,C 180,E1 -23551.565,E2 -23551.565} C_VEL
LIN {X 0,Y 157.299,Z 310.694,A -85,B 0,C 180,E1 -23556.29,E2 -23556.29} C_VEL
LIN {X 0,Y 157.404,Z 310.688,A -85,B 0,C 180,E1 -23561.788,E2 -23561.788} C_VEL
LIN {X 0,Y 157.52,Z 310.674,A -85,B 0,C 180,E1 -23567.11,E2 -23567.11} C_VEL
LIN {X 0,Y 157.685,Z 310.634,A -85,B 0,C 180,E1 -23569.731,E2 -23569.731} C_VEL
LIN {X 0,Y 157.764,Z 310.629,A -85,B 0,C 180,E1 -23572.32,E2 -23572.32} C_VEL
LIN {X 0,Y 158.25,Z 310.58,A -85,B 0,C 180,E1 -23580,E2 -23580} C_VEL
LIN {X 0,Y 158.042,Z 310.604,A -85,B 0,C 180,E1 -23581.832,E2 -23581.832} C_VEL
LIN {X 0,Y 158.701,Z 313.086,A -85,B 0,C 180,E1 -23582.935,E2 -23582.935} C_VEL
LIN {X 0,Y 160.363,Z 315.35,A -85,B 0,C 180,E1 -23584.871,E2 -23584.871} C_VEL
LIN {X 0,Y 162.561,Z 316.644,A -85,B 0,C 180,E1 -23586.891,E2 -23586.891} C_VEL
LIN {X 0,Y 164.158,Z 319.659,A -85,B 0,C 180,E1 -23588.463,E2 -23588.463} C_VEL
LIN {X 0,Y 166.634,Z 322.115,A -85,B 0,C 180,E1 -23590.423,E2 -23590.423} C_VEL
LIN {X 0,Y 168.811,Z 325.509,A -85,B 0,C 180,E1 -23592.091,E2 -23592.091} C_VEL
LIN {X 0,Y 170.426,Z 327.298,A -85,B 0,C 180,E1 -23593.185,E2 -23593.185} C_VEL
LIN {X 0,Y 173.22,Z 331.151,A -85,B 0,C 180,E1 -23595.001,E2 -23595.001} C_VEL
LIN {X 0,Y 179.096,Z 339.915,A -85,B 0,C 180,E1 -23598.376,E2 -23598.376} C_VEL
LIN {X 0,Y 183.897,Z 347.967,A -85,B 0,C 180,E1 -23600.816,E2 -23600.816} C_VEL
LIN {X 0,Y 187.277,Z 354.769,A -85,B 0,C 180,E1 -23602.449,E2 -23602.449} C_VEL
LIN {X 0,Y 188.855,Z 358.684,A -85,B 0,C 180,E1 -23603.22,E2 -23603.22} C_VEL
LIN {X 0,Y 186.966,Z 383.22,A -85,B 0,C 180,E1 -23604.2,E2 -23604.2} C_VEL
LIN {X 0,Y 185.229,Z 395.511,A -85,B 0,C 180,E1 -23605.063,E2 -23605.063} C_VEL
LIN {X 0,Y 183.077,Z 405.797,A -85,B 0,C 180,E1 -23606.195,E2 -23606.195} C_VEL
LIN {X 0,Y 180.405,Z 415.515,A -85,B 0,C 180,E1 -23607.618,E2 -23607.618} C_VEL
LIN {X 0,Y 177.375,Z 424.545,A -85,B 0,C 180,E1 -23609.348,E2 -23609.348} C_VEL
LIN {X 0,Y 173.596,Z 434.028,A -85,B 0,C 180,E1 -23611.772,E2 -23611.772} C_VEL
LIN {X 0,Y 170.077,Z 441.413,A -85,B 0,C 180,E1 -23614.267,E2 -23614.267} C_VEL
LIN {X 0,Y 166.865,Z 447.388,A -85,B 0,C 180,E1 -23616.85,E2 -23616.85} C_VEL
LIN {X 0,Y 164.072,Z 452.239,A -85,B 0,C 180,E1 -23619.556,E2 -23619.556} C_VEL
LIN {X 0,Y 161.671,Z 456.109,A -85,B 0,C 180,E1 -23622.355,E2 -23622.355} C_VEL
LIN {X 0,Y 159.554,Z 459.097,A -85,B 0,C 180,E1 -23625.191,E2 -23625.191} C_VEL
LIN {X 0,Y 157.877,Z 461.317,A -85,B 0,C 180,E1 -23628.109,E2 -23628.109} C_VEL
LIN {X 0,Y 156.514,Z 462.82,A -85,B 0,C 180,E1 -23631.051,E2 -23631.051} C_VEL
LIN {X 0,Y 155.381,Z 463.7,A -85,B 0,C 180,E1 -23634.504,E2 -23634.504} C_VEL
LIN {X 0,Y 154.812,Z 463.826,A -85,B 0,C 180,E1 -23636.993,E2 -23636.993} C_VEL
LIN {X 0,Y 154.467,Z 463.357,A -85,B 0,C 180,E1 -23639.969,E2 -23639.969} C_VEL
LIN {X 0,Y 154.379,Z 462.222,A -85,B 0,C 180,E1 -23642.92,E2 -23642.92} C_VEL
LIN {X 0,Y 154.84,Z 459.229,A -85,B 0,C 180,E1 -23647.307,E2 -23647.307} C_VEL
LIN {X 0,Y 155.735,Z 454.995,A -85,B 0,C 180,E1 -23651.386,E2 -23651.386} C_VEL
LIN {X 0,Y 156.872,Z 449.779,A -85,B 0,C 180,E1 -23655.072,E2 -23655.072} C_VEL
LIN {X 0,Y 158.562,Z 442.846,A -85,B 0,C 180,E1 -23658.691,E2 -23658.691} C_VEL
LIN {X 0,Y 160.019,Z 436.861,A -85,B 0,C 180,E1 -23661.158,E2 -23661.158} C_VEL
LIN {X 0,Y 161.706,Z 429.562,A -85,B 0,C 180,E1 -23663.59,E2 -23663.59} C_VEL
LIN {X 0,Y 163.427,Z 421.736,A -85,B 0,C 180,E1 -23665.684,E2 -23665.684} C_VEL
LIN {X 0,Y 164.893,Z 414.485,A -85,B 0,C 180,E1 -23667.252,E2 -23667.252} C_VEL
LIN {X 0,Y 166.431,Z 405.555,A -85,B 0,C 180,E1 -23668.79,E2 -23668.79} C_VEL
LIN {X 0,Y 167.753,Z 395.19,A -85,B 0,C 180,E1 -23670.153,E2 -23670.153} C_VEL
LIN {X 0,Y 168.904,Z 383.799,A -85,B 0,C 180,E1 -23671.148,E2 -23671.148} C_VEL
LIN {X 0,Y 169.933,Z 364.378,A -85,B 0,C 180,E1 -23672.077,E2 -23672.077} C_VEL
LIN {X 0,Y 170.928,Z 342.803,A -85,B 0,C 180,E1 -23672.992,E2 -23672.992} C_VEL
LIN {X 0,Y 166.334,Z 328.687,A -85,B 0,C 180,E1 -23674.43,E2 -23674.43} C_VEL
LIN {X 0,Y 157.939,Z 311.531,A -85,B 0,C 180,E1 -23676.834,E2 -23676.834} C_VEL
LIN {X 0,Y 157.769,Z 310.64,A -85,B 0,C 180,E1 -23677.037,E2 -23677.037} C_VEL
LIN {X 0,Y 157.635,Z 310.65,A -85,B 0,C 180,E1 -23681.229,E2 -23681.229} C_VEL
LIN {X 0,Y 157.436,Z 310.685,A -85,B 0,C 180,E1 -23685.535,E2 -23685.535} C_VEL
LIN {X 0,Y 157.367,Z 310.665,A -85,B 0,C 180,E1 -23690.933,E2 -23690.933} C_VEL
LIN {X 0,Y 157.31,Z 310.704,A -85,B 0,C 180,E1 -23696.68,E2 -23696.68} C_VEL
LIN {X 0,Y 157.281,Z 310.697,A -85,B 0,C 180,E1 -23702.425,E2 -23702.425} C_VEL
LIN {X 0,Y 157.268,Z 310.708,A -85,B 0,C 180,E1 -23706.448,E2 -23706.448} C_VEL
LIN {X 0,Y 157.21,Z 310.698,A -85,B 0,C 180,E1 -23712.109,E2 -23712.109} C_VEL
LIN {X 0,Y 157.247,Z 310.71,A -85,B 0,C 180,E1 -23717.901,E2 -23717.901} C_VEL
LIN {X 0,Y 157.32,Z 310.681,A -85,B 0,C 180,E1 -23723.523,E2 -23723.523} C_VEL
LIN {X 0,Y 157.292,Z 310.695,A -85,B 0,C 180,E1 -23728.094,E2 -23728.094} C_VEL
LIN {X 0,Y 157.314,Z 310.699,A -85,B 0,C 180,E1 -23733.464,E2 -23733.464} C_VEL
LIN {X 0,Y 157.39,Z 310.662,A -85,B 0,C 180,E1 -23739.668,E2 -23739.668} C_VEL
LIN {X 0,Y 157.448,Z 310.68,A -85,B 0,C 180,E1 -23744.465,E2 -23744.465} C_VEL
LIN {X 0,Y 157.685,Z 310.651,A -85,B 0,C 180,E1 -23749.73,E2 -23749.73} C_VEL
LIN {X 0,Y 157.762,Z 310.63,A -85,B 0,C 180,E1 -23752.319,E2 -23752.319} C_VEL
LIN {X 0,Y 158.251,Z 310.58,A -85,B 0,C 180,E1 -23760,E2 -23760} C_VEL
LIN {X 0,Y 157.762,Z 310.629,A -85,B 0,C 180,E1 -23767.68,E2 -23767.68} C_VEL
LIN {X 0,Y 157.632,Z 310.646,A -85,B 0,C 180,E1 -23771.235,E2 -23771.235} C_VEL
LIN {X 0,Y 157.436,Z 310.687,A -85,B 0,C 180,E1 -23775.536,E2 -23775.536} C_VEL
LIN {X 0,Y 157.363,Z 310.68,A -85,B 0,C 180,E1 -23780.933,E2 -23780.933} C_VEL
LIN {X 0,Y 157.306,Z 310.702,A -85,B 0,C 180,E1 -23786.681,E2 -23786.681} C_VEL
LIN {X 0,Y 157.271,Z 310.704,A -85,B 0,C 180,E1 -23792.428,E2 -23792.428} C_VEL
LIN {X 0,Y 157.264,Z 310.706,A -85,B 0,C 180,E1 -23796.45,E2 -23796.45} C_VEL
LIN {X 0,Y 157.19,Z 310.695,A -85,B 0,C 180,E1 -23802.117,E2 -23802.117} C_VEL
LIN {X 0,Y 157.19,Z 310.716,A -85,B 0,C 180,E1 -23807.884,E2 -23807.884} C_VEL
LIN {X 0,Y 157.324,Z 310.774,A -85,B 0,C 180,E1 -23813.597,E2 -23813.597} C_VEL
LIN {X 0,Y 157.684,Z 312.457,A -85,B 0,C 180,E1 -23814.775,E2 -23814.775} C_VEL
LIN {X 0,Y 164.869,Z 330.993,A -85,B 0,C 180,E1 -23817.053,E2 -23817.053} C_VEL
LIN {X 0,Y 167.606,Z 339.98,A -85,B 0,C 180,E1 -23817.957,E2 -23817.957} C_VEL
LIN {X 0,Y 170.144,Z 363.997,A -85,B 0,C 180,E1 -23819.538,E2 -23819.538} C_VEL
LIN {X 0,Y 168.871,Z 390.164,A -85,B 0,C 180,E1 -23820.725,E2 -23820.725} C_VEL
LIN {X 0,Y 167.885,Z 400.526,A -85,B 0,C 180,E1 -23821.504,E2 -23821.504} C_VEL
LIN {X 0,Y 166.277,Z 411.844,A -85,B 0,C 180,E1 -23822.798,E2 -23822.798} C_VEL
LIN {X 0,Y 164.748,Z 421.583,A -85,B 0,C 180,E1 -23824.411,E2 -23824.411} C_VEL
LIN {X 0,Y 162.881,Z 429.882,A -85,B 0,C 180,E1 -23826.14,E2 -23826.14} C_VEL
LIN {X 0,Y 161.497,Z 436.789,A -85,B 0,C 180,E1 -23827.955,E2 -23827.955} C_VEL
LIN {X 0,Y 159.875,Z 443.485,A -85,B 0,C 180,E1 -23830.082,E2 -23830.082} C_VEL
LIN {X 0,Y 158.293,Z 449.839,A -85,B 0,C 180,E1 -23832.561,E2 -23832.561} C_VEL
LIN {X 0,Y 157.078,Z 455.118,A -85,B 0,C 180,E1 -23835.092,E2 -23835.092} C_VEL
LIN {X 0,Y 155.915,Z 460.47,A -85,B 0,C 180,E1 -23838.297,E2 -23838.297} C_VEL
LIN {X 0,Y 155.308,Z 463.906,A -85,B 0,C 180,E1 -23840.887,E2 -23840.887} C_VEL
LIN {X 0,Y 154.911,Z 466.694,A -85,B 0,C 180,E1 -23843.488,E2 -23843.488} C_VEL
LIN {X 0,Y 154.741,Z 469.891,A -85,B 0,C 180,E1 -23847.69,E2 -23847.69} C_VEL
LIN {X 0,Y 154.824,Z 471.053,A -85,B 0,C 180,E1 -23850,E2 -23850} C_VEL
LIN {X 0,Y 154.698,Z 471.896,A -85,B 0,C 180,E1 -23852.604,E2 -23852.604} C_VEL
LIN {X 0,Y 154.789,Z 472.174,A -85,B 0,C 180,E1 -23855.21,E2 -23855.21} C_VEL
LIN {X 0,Y 154.993,Z 471.975,A -85,B 0,C 180,E1 -23857.274,E2 -23857.274} C_VEL
LIN {X 0,Y 154.746,Z 471.6,A -85,B 0,C 180,E1 -23859.45,E2 -23859.45} C_VEL
LIN {X 0,Y 152.987,Z 470.207,A -85,B 0,C 180,E1 -23863.046,E2 -23863.046} C_VEL
LIN {X 0,Y 151.758,Z 468.065,A -85,B 0,C 180,E1 -23866.658,E2 -23866.658} C_VEL
LIN {X 0,Y 152.34,Z 466.256,A -85,B 0,C 180,E1 -23868.78,E2 -23868.78} C_VEL
LIN {X 0,Y 155.369,Z 461.915,A -85,B 0,C 180,E1 -23872.611,E2 -23872.611} C_VEL
LIN {X 0,Y 159.018,Z 456.035,A -85,B 0,C 180,E1 -23876.228,E2 -23876.228} C_VEL
LIN {X 0,Y 161.85,Z 451.179,A -85,B 0,C 180,E1 -23878.531,E2 -23878.531} C_VEL
LIN {X 0,Y 164.948,Z 445.349,A -85,B 0,C 180,E1 -23880.748,E2 -23880.748} C_VEL
LIN {X 0,Y 168.177,Z 438.3,A -85,B 0,C 180,E1 -23882.905,E2 -23882.905} C_VEL
LIN {X 0,Y 171.412,Z 430.669,A -85,B 0,C 180,E1 -23884.716,E2 -23884.716} C_VEL
LIN {X 0,Y 174.237,Z 422.764,A -85,B 0,C 180,E1 -23886.224,E2 -23886.224} C_VEL
LIN {X 0,Y 176.641,Z 415.142,A -85,B 0,C 180,E1 -23887.353,E2 -23887.353} C_VEL
LIN {X 0,Y 178.997,Z 406.076,A -85,B 0,C 180,E1 -23888.377,E2 -23888.377} C_VEL
LIN {X 0,Y 180.864,Z 396.534,A -85,B 0,C 180,E1 -23889.168,E2 -23889.168} C_VEL
LIN {X 0,Y 182.221,Z 386.21,A -85,B 0,C 180,E1 -23889.739,E2 -23889.739} C_VEL
LIN {X 0,Y 183.346,Z 369.711,A -85,B 0,C 180,E1 -23890.435,E2 -23890.435} C_VEL
LIN {X 0,Y 182.896,Z 365.356,A -85,B 0,C 180,E1 -23890.876,E2 -23890.876} C_VEL
LIN {X 0,Y 178.722,Z 354.841,A -85,B 0,C 180,E1 -23893.172,E2 -23893.172} C_VEL
LIN {X 0,Y 174.752,Z 346.602,A -85,B 0,C 180,E1 -23895.505,E2 -23895.505} C_VEL
LIN {X 0,Y 171.556,Z 340.804,A -85,B 0,C 180,E1 -23897.508,E2 -23897.508} C_VEL
LIN {X 0,Y 169.545,Z 337.347,A -85,B 0,C 180,E1 -23898.871,E2 -23898.871} C_VEL
LIN {X 0,Y 167.068,Z 333.19,A -85,B 0,C 180,E1 -23900.693,E2 -23900.693} C_VEL
LIN {X 0,Y 164.024,Z 328.349,A -85,B 0,C 180,E1 -23903.14,E2 -23903.14} C_VEL
LIN {X 0,Y 161.498,Z 325.896,A -85,B 0,C 180,E1 -23905.319,E2 -23905.319} C_VEL
LIN {X 0,Y 160.092,Z 323.239,A -85,B 0,C 180,E1 -23906.813,E2 -23906.813} C_VEL
LIN {X 0,Y 157.443,Z 321.162,A -85,B 0,C 180,E1 -23909.622,E2 -23909.622} C_VEL
LIN {X 0,Y 155.886,Z 318.539,A -85,B 0,C 180,E1 -23911.838,E2 -23911.838} C_VEL
LIN {X 0,Y 155.566,Z 317.564,A -85,B 0,C 180,E1 -23912.415,E2 -23912.415} C_VEL
LIN {X 0,Y 152.299,Z 315.71,A -85,B 0,C 180,E1 -23918.336,E2 -23918.336} C_VEL
LIN {X 0,Y 151.011,Z 313.689,A -85,B 0,C 180,E1 -23924.479,E2 -23924.479} C_VEL
LIN {X 0,Y 151.018,Z 313.452,A -85,B 0,C 180,E1 -23927.757,E2 -23927.757} C_VEL
LIN {X 0,Y 151.483,Z 314.053,A -85,B 0,C 180,E1 -23930.992,E2 -23930.992} C_VEL
LIN {X 0,Y 154.484,Z 316.741,A -85,B 0,C 180,E1 -23938.403,E2 -23938.403} C_VEL
LIN {X 0,Y 156.295,Z 317.641,A -85,B 0,C 180,E1 -23940.967,E2 -23940.967} C_VEL
LIN {X 0,Y 157.438,Z 320.454,A -85,B 0,C 180,E1 -23942.719,E2 -23942.719} C_VEL
LIN {X 0,Y 159.503,Z 322.632,A -85,B 0,C 180,E1 -23945.056,E2 -23945.056} C_VEL
LIN {X 0,Y 160.619,Z 323.422,A -85,B 0,C 180,E1 -23946.123,E2 -23946.123} C_VEL
LIN {X 0,Y 162.652,Z 326.72,A -85,B 0,C 180,E1 -23948.134,E2 -23948.134} C_VEL
LIN {X 0,Y 164.405,Z 328.595,A -85,B 0,C 180,E1 -23949.613,E2 -23949.613} C_VEL
LIN {X 0,Y 166.823,Z 332.164,A -85,B 0,C 180,E1 -23951.521,E2 -23951.521} C_VEL
LIN {X 0,Y 168.11,Z 333.825,A -85,B 0,C 180,E1 -23952.449,E2 -23952.449} C_VEL
LIN {X 0,Y 171.345,Z 338.511,A -85,B 0,C 180,E1 -23954.661,E2 -23954.661} C_VEL
LIN {X 0,Y 175.967,Z 345.625,A -85,B 0,C 180,E1 -23957.431,E2 -23957.431} C_VEL
LIN {X 0,Y 180.195,Z 352.985,A -85,B 0,C 180,E1 -23959.748,E2 -23959.748} C_VEL
LIN {X 0,Y 183.281,Z 359.417,A -85,B 0,C 180,E1 -23961.337,E2 -23961.337} C_VEL
LIN {X 0,Y 183.963,Z 361.222,A -85,B 0,C 180,E1 -23961.699,E2 -23961.699} C_VEL
LIN {X 0,Y 182.111,Z 383.647,A -85,B 0,C 180,E1 -23962.606,E2 -23962.606} C_VEL
LIN {X 0,Y 180.313,Z 395.624,A -85,B 0,C 180,E1 -23963.453,E2 -23963.453} C_VEL
LIN {X 0,Y 177.885,Z 406.533,A -85,B 0,C 180,E1 -23964.678,E2 -23964.678} C_VEL
LIN {X 0,Y 175.711,Z 414.19,A -85,B 0,C 180,E1 -23965.796,E2 -23965.796} C_VEL
LIN {X 0,Y 172.941,Z 422.2,A -85,B 0,C 180,E1 -23967.261,E2 -23967.261} C_VEL
LIN {X 0,Y 169.882,Z 429.952,A -85,B 0,C 180,E1 -23969.083,E2 -23969.083} C_VEL
LIN {X 0,Y 166.451,Z 437.497,A -85,B 0,C 180,E1 -23971.333,E2 -23971.333} C_VEL
LIN {X 0,Y 162.072,Z 445.686,A -85,B 0,C 180,E1 -23974.525,E2 -23974.525} C_VEL
LIN {X 0,Y 158.91,Z 450.876,A -85,B 0,C 180,E1 -23977.246,E2 -23977.246} C_VEL
LIN {X 0,Y 156.198,Z 455.075,A -85,B 0,C 180,E1 -23980.104,E2 -23980.104} C_VEL
LIN {X 0,Y 153.529,Z 458.678,A -85,B 0,C 180,E1 -23983.366,E2 -23983.366} C_VEL
LIN {X 0,Y 151.797,Z 460.869,A -85,B 0,C 180,E1 -23986.016,E2 -23986.016} C_VEL
LIN {X 0,Y 150.205,Z 462.636,A -85,B 0,C 180,E1 -23989.078,E2 -23989.078} C_VEL
LIN {X 0,Y 148.5,Z 463.881,A -85,B 0,C 180,E1 -23993.568,E2 -23993.568} C_VEL
LIN {X 0,Y 148.065,Z 464.058,A -85,B 0,C 180,E1 -23995.28,E2 -23995.28} C_VEL
LIN {X 0,Y 147.45,Z 463.669,A -85,B 0,C 180,E1 -23999.087,E2 -23999.087} C_VEL
LIN {X 0,Y 147.272,Z 462.847,A -85,B 0,C 180,E1 -24001.497,E2 -24001.497} C_VEL
LIN {X 0,Y 147.585,Z 460.21,A -85,B 0,C 180,E1 -24006.298,E2 -24006.298} C_VEL
LIN {X 0,Y 148.107,Z 457.763,A -85,B 0,C 180,E1 -24009.153,E2 -24009.153} C_VEL
LIN {X 0,Y 149.236,Z 452.542,A -85,B 0,C 180,E1 -24013.588,E2 -24013.588} C_VEL
LIN {X 0,Y 150.267,Z 448.095,A -85,B 0,C 180,E1 -24016.477,E2 -24016.477} C_VEL
LIN {X 0,Y 151.656,Z 442.657,A -85,B 0,C 180,E1 -24019.318,E2 -24019.318} C_VEL
LIN {X 0,Y 153.327,Z 436.036,A -85,B 0,C 180,E1 -24022.097,E2 -24022.097} C_VEL
LIN {X 0,Y 154.829,Z 429.901,A -85,B 0,C 180,E1 -24024.204,E2 -24024.204} C_VEL
LIN {X 0,Y 156.397,Z 423.1,A -85,B 0,C 180,E1 -24026.135,E2 -24026.135} C_VEL
LIN {X 0,Y 158.216,Z 414.492,A -85,B 0,C 180,E1 -24028.091,E2 -24028.091} C_VEL
LIN {X 0,Y 159.812,Z 405.524,A -85,B 0,C 180,E1 -24029.685,E2 -24029.685} C_VEL
LIN {X 0,Y 161.168,Z 395.381,A -85,B 0,C 180,E1 -24031.06,E2 -24031.06} C_VEL
LIN {X 0,Y 162.412,Z 383.383,A -85,B 0,C 180,E1 -24032.124,E2 -24032.124} C_VEL
LIN {X 0,Y 163.534,Z 362.511,A -85,B 0,C 180,E1 -24033.14,E2 -24033.14} C_VEL
LIN {X 0,Y 164.357,Z 344.123,A -85,B 0,C 180,E1 -24033.959,E2 -24033.959} C_VEL
LIN {X 0,Y 160.446,Z 331.85,A -85,B 0,C 180,E1 -24035.275,E2 -24035.275} C_VEL
LIN {X 0,Y 151.58,Z 314.158,A -85,B 0,C 180,E1 -24037.944,E2 -24037.944} C_VEL
LIN {X 0,Y 150.685,Z 311.529,A -85,B 0,C 180,E1 -24038.296,E2 -24038.296} C_VEL
LIN {X 0,Y 150.576,Z 311.527,A -85,B 0,C 180,E1 -24041.432,E2 -24041.432} C_VEL
LIN {X 0,Y 150.346,Z 311.571,A -85,B 0,C 180,E1 -24046.288,E2 -24046.288} C_VEL
LIN {X 0,Y 150.349,Z 311.539,A -85,B 0,C 180,E1 -24050.789,E2 -24050.789} C_VEL
LIN {X 0,Y 150.242,Z 311.588,A -85,B 0,C 180,E1 -24057.279,E2 -24057.279} C_VEL
LIN {X 0,Y 150.22,Z 311.576,A -85,B 0,C 180,E1 -24062.634,E2 -24062.634} C_VEL
LIN {X 0,Y 150.177,Z 311.593,A -85,B 0,C 180,E1 -24067.471,E2 -24067.471} C_VEL
LIN {X 0,Y 150.15,Z 311.579,A -85,B 0,C 180,E1 -24071.504,E2 -24071.504} C_VEL
LIN {X 0,Y 150.174,Z 311.585,A -85,B 0,C 180,E1 -24075.413,E2 -24075.413} C_VEL
LIN {X 0,Y 150.206,Z 311.587,A -85,B 0,C 180,E1 -24079.076,E2 -24079.076} C_VEL
LIN {X 0,Y 150.233,Z 311.571,A -85,B 0,C 180,E1 -24082.679,E2 -24082.679} C_VEL
LIN {X 0,Y 150.215,Z 311.573,A -85,B 0,C 180,E1 -24087.365,E2 -24087.365} C_VEL
LIN {X 0,Y 150.239,Z 311.581,A -85,B 0,C 180,E1 -24092.719,E2 -24092.719} C_VEL
LIN {X 0,Y 150.347,Z 311.538,A -85,B 0,C 180,E1 -24099.208,E2 -24099.208} C_VEL
LIN {X 0,Y 150.357,Z 311.561,A -85,B 0,C 180,E1 -24103.712,E2 -24103.712} C_VEL
LIN {X 0,Y 150.607,Z 311.533,A -85,B 0,C 180,E1 -24109.242,E2 -24109.242} C_VEL
LIN {X 0,Y 150.7,Z 311.512,A -85,B 0,C 180,E1 -24111.957,E2 -24111.957} C_VEL
LIN {X 0,Y 151.212,Z 311.457,A -85,B 0,C 180,E1 -24120,E2 -24120} C_VEL
LIN {X 0,Y 150.699,Z 311.507,A -85,B 0,C 180,E1 -24128.042,E2 -24128.042} C_VEL
LIN {X 0,Y 150.573,Z 311.526,A -85,B 0,C 180,E1 -24131.436,E2 -24131.436} C_VEL
LIN {X 0,Y 150.347,Z 311.568,A -85,B 0,C 180,E1 -24136.288,E2 -24136.288} C_VEL
LIN {X 0,Y 150.345,Z 311.553,A -85,B 0,C 180,E1 -24140.79,E2 -24140.79} C_VEL
LIN {X 0,Y 150.237,Z 311.582,A -85,B 0,C 180,E1 -24147.28,E2 -24147.28} C_VEL
LIN {X 0,Y 150.211,Z 311.585,A -85,B 0,C 180,E1 -24152.632,E2 -24152.632} C_VEL
LIN {X 0,Y 150.169,Z 311.585,A -85,B 0,C 180,E1 -24157.474,E2 -24157.474} C_VEL
LIN {X 0,Y 150.133,Z 311.569,A -85,B 0,C 180,E1 -24161.499,E2 -24161.499} C_VEL
LIN {X 0,Y 150.124,Z 311.597,A -85,B 0,C 180,E1 -24165.396,E2 -24165.396} C_VEL
LIN {X 0,Y 150.139,Z 311.597,A -85,B 0,C 180,E1 -24169.056,E2 -24169.056} C_VEL
LIN {X 0,Y 150.24,Z 311.699,A -85,B 0,C 180,E1 -24172.919,E2 -24172.919} C_VEL
LIN {X 0,Y 150.38,Z 312.274,A -85,B 0,C 180,E1 -24173.301,E2 -24173.301} C_VEL
LIN {X 0,Y 157.28,Z 329.416,A -85,B 0,C 180,E1 -24175.628,E2 -24175.628} C_VEL
LIN {X 0,Y 161.212,Z 341.094,A -85,B 0,C 180,E1 -24176.961,E2 -24176.961} C_VEL
LIN {X 0,Y 163.594,Z 365.06,A -85,B 0,C 180,E1 -24178.605,E2 -24178.605} C_VEL
LIN {X 0,Y 162.258,Z 391.03,A -85,B 0,C 180,E1 -24179.842,E2 -24179.842} C_VEL
LIN {X 0,Y 161.118,Z 401.749,A -85,B 0,C 180,E1 -24180.708,E2 -24180.708} C_VEL
LIN {X 0,Y 159.558,Z 412.1,A -85,B 0,C 180,E1 -24181.994,E2 -24181.994} C_VEL
LIN {X 0,Y 158.045,Z 421.396,A -85,B 0,C 180,E1 -24183.598,E2 -24183.598} C_VEL
LIN {X 0,Y 156.102,Z 429.692,A -85,B 0,C 180,E1 -24185.39,E2 -24185.39} C_VEL
LIN {X 0,Y 154.378,Z 437.621,A -85,B 0,C 180,E1 -24187.588,E2 -24187.588} C_VEL
LIN {X 0,Y 152.742,Z 444.152,A -85,B 0,C 180,E1 -24189.813,E2 -24189.813} C_VEL
LIN {X 0,Y 151.152,Z 450.365,A -85,B 0,C 180,E1 -24192.409,E2 -24192.409} C_VEL
LIN {X 0,Y 149.921,Z 455.52,A -85,B 0,C 180,E1 -24195.059,E2 -24195.059} C_VEL
LIN {X 0,Y 148.958,Z 459.796,A -85,B 0,C 180,E1 -24197.742,E2 -24197.742} C_VEL
LIN {X 0,Y 148.292,Z 463.33,A -85,B 0,C 180,E1 -24200.452,E2 -24200.452} C_VEL
LIN {X 0,Y 147.72,Z 467.366,A -85,B 0,C 180,E1 -24204.54,E2 -24204.54} C_VEL
LIN {X 0,Y 147.65,Z 469.934,A -85,B 0,C 180,E1 -24208.329,E2 -24208.329} C_VEL
LIN {X 0,Y 147.633,Z 471.22,A -85,B 0,C 180,E1 -24211.432,E2 -24211.432} C_VEL
LIN {X 0,Y 147.715,Z 471.936,A -85,B 0,C 180,E1 -24215.46,E2 -24215.46} C_VEL
LIN {X 0,Y 148.035,Z 471.763,A -85,B 0,C 180,E1 -24218.188,E2 -24218.188} C_VEL
LIN {X 0,Y 148.649,Z 471.145,A -85,B 0,C 180,E1 -24220.901,E2 -24220.901} C_VEL
LIN {X 0,Y 149.602,Z 470.071,A -85,B 0,C 180,E1 -24223.585,E2 -24223.585} C_VEL
LIN {X 0,Y 151.58,Z 467.371,A -85,B 0,C 180,E1 -24227.539,E2 -24227.539} C_VEL
LIN {X 0,Y 152.34,Z 466.256,A -85,B 0,C 180,E1 -24228.78,E2 -24228.78} C_VEL
LIN {X 0,Y 153.108,Z 464.284,A -85,B 0,C 180,E1 -24230.856,E2 -24230.856} C_VEL
LIN {X 0,Y 153.05,Z 460.484,A -85,B 0,C 180,E1 -24234.298,E2 -24234.298} C_VEL
LIN {X 0,Y 153.521,Z 455.935,A -85,B 0,C 180,E1 -24237.577,E2 -24237.577} C_VEL
LIN {X 0,Y 155.055,Z 452.7,A -85,B 0,C 180,E1 -24239.323,E2 -24239.323} C_VEL
LIN {X 0,Y 159.801,Z 444.427,A -85,B 0,C 180,E1 -24242.597,E2 -24242.597} C_VEL
LIN {X 0,Y 163.149,Z 437.483,A -85,B 0,C 180,E1 -24244.721,E2 -24244.721} C_VEL
LIN {X 0,Y 166.094,Z 430.843,A -85,B 0,C 180,E1 -24246.325,E2 -24246.325} C_VEL
LIN {X 0,Y 168.815,Z 423.762,A -85,B 0,C 180,E1 -24247.722,E2 -24247.722} C_VEL
LIN {X 0,Y 171.657,Z 415.264,A -85,B 0,C 180,E1 -24249.011,E2 -24249.011} C_VEL
LIN {X 0,Y 174.103,Z 406.292,A -85,B 0,C 180,E1 -24250.04,E2 -24250.04} C_VEL
LIN {X 0,Y 176.06,Z 396.783,A -85,B 0,C 180,E1 -24250.845,E2 -24250.845} C_VEL
LIN {X 0,Y 177.373,Z 387.539,A -85,B 0,C 180,E1 -24251.379,E2 -24251.379} C_VEL
LIN {X 0,Y 178.635,Z 370.719,A -85,B 0,C 180,E1 -24252.112,E2 -24252.112} C_VEL
LIN {X 0,Y 178.373,Z 368.391,A -85,B 0,C 180,E1 -24252.373,E2 -24252.373} C_VEL
LIN {X 0,Y 174.59,Z 358.521,A -85,B 0,C 180,E1 -24254.672,E2 -24254.672} C_VEL
LIN {X 0,Y 170.067,Z 349.025,A -85,B 0,C 180,E1 -24257.583,E2 -24257.583} C_VEL
LIN {X 0,Y 166.754,Z 343.017,A -85,B 0,C 180,E1 -24259.955,E2 -24259.955} C_VEL
LIN {X 0,Y 164.267,Z 338.806,A -85,B 0,C 180,E1 -24261.903,E2 -24261.903} C_VEL
LIN {X 0,Y 161.713,Z 334.681,A -85,B 0,C 180,E1 -24264.126,E2 -24264.126} C_VEL
LIN {X 0,Y 159.122,Z 331.669,A -85,B 0,C 180,E1 -24266.575,E2 -24266.575} C_VEL
LIN {X 0,Y 158.069,Z 329.806,A -85,B 0,C 180,E1 -24267.756,E2 -24267.756} C_VEL
LIN {X 0,Y 155.474,Z 327.315,A -85,B 0,C 180,E1 -24270.834,E2 -24270.834} C_VEL
LIN {X 0,Y 153.965,Z 324.41,A -85,B 0,C 180,E1 -24273.258,E2 -24273.258} C_VEL
LIN {X 0,Y 150.894,Z 322.245,A -85,B 0,C 180,E1 -24279.625,E2 -24279.625} C_VEL
LIN {X 0,Y 150.017,Z 320.609,A -85,B 0,C 180,E1 -24285.069,E2 -24285.069} C_VEL
LIN {X 0,Y 150.321,Z 320.776,A -85,B 0,C 180,E1 -24289.901,E2 -24289.901} C_VEL
LIN {X 0,Y 153.484,Z 323.789,A -85,B 0,C 180,E1 -24298.402,E2 -24298.402} C_VEL
LIN {X 0,Y 154.671,Z 324.411,A -85,B 0,C 180,E1 -24300.147,E2 -24300.147} C_VEL
LIN {X 0,Y 156.119,Z 327.566,A -85,B 0,C 180,E1 -24302.399,E2 -24302.399} C_VEL
LIN {X 0,Y 158.778,Z 330.163,A -85,B 0,C 180,E1 -24305.397,E2 -24305.397} C_VEL
LIN {X 0,Y 161.05,Z 333.571,A -85,B 0,C 180,E1 -24307.696,E2 -24307.696} C_VEL
LIN {X 0,Y 162.301,Z 335.139,A -85,B 0,C 180,E1 -24308.82,E2 -24308.82} C_VEL
LIN {X 0,Y 164.949,Z 338.904,A -85,B 0,C 180,E1 -24311.008,E2 -24311.008} C_VEL
LIN {X 0,Y 168.83,Z 344.795,A -85,B 0,C 180,E1 -24313.849,E2 -24313.849} C_VEL
LIN {X 0,Y 173.622,Z 352.548,A -85,B 0,C 180,E1 -24316.891,E2 -24316.891} C_VEL
LIN {X 0,Y 177.791,Z 360.35,A -85,B 0,C 180,E1 -24319.296,E2 -24319.296} C_VEL
LIN {X 0,Y 179.185,Z 363.636,A -85,B 0,C 180,E1 -24320.082,E2 -24320.082} C_VEL
LIN {X 0,Y 177.345,Z 384.465,A -85,B 0,C 180,E1 -24320.937,E2 -24320.937} C_VEL
LIN {X 0,Y 175.247,Z 397.114,A -85,B 0,C 180,E1 -24321.888,E2 -24321.888} C_VEL
LIN {X 0,Y 173.129,Z 406.284,A -85,B 0,C 180,E1 -24322.937,E2 -24322.937} C_VEL
LIN {X 0,Y 170.446,Z 415.193,A -85,B 0,C 180,E1 -24324.255,E2 -24324.255} C_VEL
LIN {X 0,Y 167.656,Z 422.79,A -85,B 0,C 180,E1 -24325.68,E2 -24325.68} C_VEL
LIN {X 0,Y 164.836,Z 429.621,A -85,B 0,C 180,E1 -24327.305,E2 -24327.305} C_VEL
LIN {X 0,Y 161.394,Z 436.823,A -85,B 0,C 180,E1 -24329.438,E2 -24329.438} C_VEL
LIN {X 0,Y 157.543,Z 443.773,A -85,B 0,C 180,E1 -24332.052,E2 -24332.052} C_VEL
LIN {X 0,Y 153.334,Z 450.495,A -85,B 0,C 180,E1 -24335.414,E2 -24335.414} C_VEL
LIN {X 0,Y 149.585,Z 455.782,A -85,B 0,C 180,E1 -24339.177,E2 -24339.177} C_VEL
LIN {X 0,Y 147.301,Z 458.696,A -85,B 0,C 180,E1 -24341.911,E2 -24341.911} C_VEL
LIN {X 0,Y 145.936,Z 460.26,A -85,B 0,C 180,E1 -24343.751,E2 -24343.751} C_VEL
LIN {X 0,Y 143.986,Z 462.332,A -85,B 0,C 180,E1 -24347.068,E2 -24347.068} C_VEL
LIN {X 0,Y 142.54,Z 463.533,A -85,B 0,C 180,E1 -24350.137,E2 -24350.137} C_VEL
LIN {X 0,Y 141.411,Z 464.147,A -85,B 0,C 180,E1 -24353.39,E2 -24353.39} C_VEL
LIN {X 0,Y 140.423,Z 463.909,A -85,B 0,C 180,E1 -24358.302,E2 -24358.302} C_VEL
LIN {X 0,Y 140.169,Z 462.155,A -85,B 0,C 180,E1 -24363.177,E2 -24363.177} C_VEL
LIN {X 0,Y 140.515,Z 460.198,A -85,B 0,C 180,E1 -24366.415,E2 -24366.415} C_VEL
LIN {X 0,Y 141.079,Z 457.555,A -85,B 0,C 180,E1 -24369.592,E2 -24369.592} C_VEL
LIN {X 0,Y 142.038,Z 453.194,A -85,B 0,C 180,E1 -24373.471,E2 -24373.471} C_VEL
LIN {X 0,Y 143.299,Z 448.033,A -85,B 0,C 180,E1 -24376.984,E2 -24376.984} C_VEL
LIN {X 0,Y 144.892,Z 441.98,A -85,B 0,C 180,E1 -24380.226,E2 -24380.226} C_VEL
LIN {X 0,Y 146.232,Z 437.029,A -85,B 0,C 180,E1 -24382.405,E2 -24382.405} C_VEL
LIN {X 0,Y 148.132,Z 429.542,A -85,B 0,C 180,E1 -24385.093,E2 -24385.093} C_VEL
LIN {X 0,Y 149.976,Z 421.806,A -85,B 0,C 180,E1 -24387.314,E2 -24387.314} C_VEL
LIN {X 0,Y 151.923,Z 412.876,A -85,B 0,C 180,E1 -24389.337,E2 -24389.337} C_VEL
LIN {X 0,Y 153.797,Z 402.139,A -85,B 0,C 180,E1 -24391.191,E2 -24391.191} C_VEL
LIN {X 0,Y 155.141,Z 391.411,A -85,B 0,C 180,E1 -24392.478,E2 -24392.478} C_VEL
LIN {X 0,Y 156.046,Z 381.478,A -85,B 0,C 180,E1 -24393.276,E2 -24393.276} C_VEL
LIN {X 0,Y 157.914,Z 345.524,A -85,B 0,C 180,E1 -24394.987,E2 -24394.987} C_VEL
LIN {X 0,Y 154.408,Z 334.562,A -85,B 0,C 180,E1 -24396.225,E2 -24396.225} C_VEL
LIN {X 0,Y 145.011,Z 315.835,A -85,B 0,C 180,E1 -24399.253,E2 -24399.253} C_VEL
LIN {X 0,Y 143.691,Z 313.01,A -85,B 0,C 180,E1 -24399.724,E2 -24399.724} C_VEL
LIN {X 0,Y 143.607,Z 312.406,A -85,B 0,C 180,E1 -24399.862,E2 -24399.862} C_VEL
LIN {X 0,Y 143.284,Z 312.448,A -85,B 0,C 180,E1 -24407.115,E2 -24407.115} C_VEL
LIN {X 0,Y 143.275,Z 312.418,A -85,B 0,C 180,E1 -24411.251,E2 -24411.251} C_VEL
LIN {X 0,Y 143.191,Z 312.465,A -85,B 0,C 180,E1 -24417.936,E2 -24417.936} C_VEL
LIN {X 0,Y 143.147,Z 312.458,A -85,B 0,C 180,E1 -24423.421,E2 -24423.421} C_VEL
LIN {X 0,Y 143.062,Z 312.472,A -85,B 0,C 180,E1 -24429.688,E2 -24429.688} C_VEL
LIN {X 0,Y 143.077,Z 312.458,A -85,B 0,C 180,E1 -24433.446,E2 -24433.446} C_VEL
LIN {X 0,Y 143.12,Z 312.469,A -85,B 0,C 180,E1 -24437.439,E2 -24437.439} C_VEL
LIN {X 0,Y 143.132,Z 312.458,A -85,B 0,C 180,E1 -24441.776,E2 -24441.776} C_VEL
LIN {X 0,Y 143.183,Z 312.448,A -85,B 0,C 180,E1 -24447.321,E2 -24447.321} C_VEL
LIN {X 0,Y 143.186,Z 312.462,A -85,B 0,C 180,E1 -24452.063,E2 -24452.063} C_VEL
LIN {X 0,Y 143.273,Z 312.419,A -85,B 0,C 180,E1 -24458.746,E2 -24458.746} C_VEL
LIN {X 0,Y 143.297,Z 312.436,A -85,B 0,C 180,E1 -24462.886,E2 -24462.886} C_VEL
LIN {X 0,Y 143.533,Z 312.417,A -85,B 0,C 180,E1 -24468.705,E2 -24468.705} C_VEL
LIN {X 0,Y 143.621,Z 312.395,A -85,B 0,C 180,E1 -24471.558,E2 -24471.558} C_VEL
LIN {X 0,Y 144.171,Z 312.334,A -85,B 0,C 180,E1 -24480,E2 -24480} C_VEL
LIN {X 0,Y 143.621,Z 312.385,A -85,B 0,C 180,E1 -24488.441,E2 -24488.441} C_VEL
LIN {X 0,Y 143.5,Z 312.407,A -85,B 0,C 180,E1 -24491.627,E2 -24491.627} C_VEL
LIN {X 0,Y 143.29,Z 312.448,A -85,B 0,C 180,E1 -24497.114,E2 -24497.114} C_VEL
LIN {X 0,Y 143.271,Z 312.433,A -85,B 0,C 180,E1 -24501.252,E2 -24501.252} C_VEL
LIN {X 0,Y 143.184,Z 312.46,A -85,B 0,C 180,E1 -24507.935,E2 -24507.935} C_VEL
LIN {X 0,Y 143.14,Z 312.468,A -85,B 0,C 180,E1 -24513.42,E2 -24513.42} C_VEL
LIN {X 0,Y 143.052,Z 312.452,A -85,B 0,C 180,E1 -24519.693,E2 -24519.693} C_VEL
LIN {X 0,Y 143.031,Z 312.468,A -85,B 0,C 180,E1 -24523.464,E2 -24523.464} C_VEL
LIN {X 0,Y 143.037,Z 312.478,A -85,B 0,C 180,E1 -24527.477,E2 -24527.477} C_VEL
LIN {X 0,Y 143.113,Z 312.471,A -85,B 0,C 180,E1 -24531.677,E2 -24531.677} C_VEL
LIN {X 0,Y 144.23,Z 315.462,A -85,B 0,C 180,E1 -24532.16,E2 -24532.16} C_VEL
LIN {X 0,Y 145.5,Z 317.814,A -85,B 0,C 180,E1 -24532.586,E2 -24532.586} C_VEL
LIN {X 0,Y 150.871,Z 331.026,A -85,B 0,C 180,E1 -24534.494,E2 -24534.494} C_VEL
LIN {X 0,Y 154.929,Z 343.024,A -85,B 0,C 180,E1 -24535.943,E2 -24535.943} C_VEL
LIN {X 0,Y 157.115,Z 364.945,A -85,B 0,C 180,E1 -24537.536,E2 -24537.536} C_VEL
LIN {X 0,Y 155.752,Z 390.941,A -85,B 0,C 180,E1 -24538.826,E2 -24538.826} C_VEL
LIN {X 0,Y 154.474,Z 402.254,A -85,B 0,C 180,E1 -24539.787,E2 -24539.787} C_VEL
LIN {X 0,Y 152.81,Z 412.701,A -85,B 0,C 180,E1 -24541.176,E2 -24541.176} C_VEL
LIN {X 0,Y 151.375,Z 421.209,A -85,B 0,C 180,E1 -24542.712,E2 -24542.712} C_VEL
LIN {X 0,Y 149.353,Z 429.502,A -85,B 0,C 180,E1 -24544.572,E2 -24544.572} C_VEL
LIN {X 0,Y 147.553,Z 437.432,A -85,B 0,C 180,E1 -24546.863,E2 -24546.863} C_VEL
LIN {X 0,Y 145.61,Z 444.82,A -85,B 0,C 180,E1 -24549.518,E2 -24549.518} C_VEL
LIN {X 0,Y 143.685,Z 452.313,A -85,B 0,C 180,E1 -24552.934,E2 -24552.934} C_VEL
LIN {X 0,Y 142.225,Z 458.154,A -85,B 0,C 180,E1 -24556.425,E2 -24556.425} C_VEL
LIN {X 0,Y 141.295,Z 462.754,A -85,B 0,C 180,E1 -24559.975,E2 -24559.975} C_VEL
LIN {X 0,Y 140.804,Z 465.721,A -85,B 0,C 180,E1 -24562.832,E2 -24562.832} C_VEL
LIN {X 0,Y 140.585,Z 468.91,A -85,B 0,C 180,E1 -24567.135,E2 -24567.135} C_VEL
LIN {X 0,Y 140.578,Z 470.715,A -85,B 0,C 180,E1 -24570.935,E2 -24570.935} C_VEL
LIN {X 0,Y 140.534,Z 471.332,A -85,B 0,C 180,E1 -24572.866,E2 -24572.866} C_VEL
LIN {X 0,Y 140.643,Z 471.695,A -85,B 0,C 180,E1 -24575.736,E2 -24575.736} C_VEL
LIN {X 0,Y 141.013,Z 471.609,A -85,B 0,C 180,E1 -24578.599,E2 -24578.599} C_VEL
LIN {X 0,Y 141.678,Z 471.078,A -85,B 0,C 180,E1 -24581.444,E2 -24581.444} C_VEL
LIN {X 0,Y 142.7,Z 470.056,A -85,B 0,C 180,E1 -24584.255,E2 -24584.255} C_VEL
LIN {X 0,Y 144.829,Z 467.484,A -85,B 0,C 180,E1 -24588.386,E2 -24588.386} C_VEL
LIN {X 0,Y 147.646,Z 463.66,A -85,B 0,C 180,E1 -24592.383,E2 -24592.383} C_VEL
LIN {X 0,Y 151.36,Z 458.483,A -85,B 0,C 180,E1 -24596.174,E2 -24596.174} C_VEL
LIN {X 0,Y 155.055,Z 452.7,A -85,B 0,C 180,E1 -24599.323,E2 -24599.323} C_VEL
LIN {X 0,Y 156.702,Z 449.279,A -85,B 0,C 180,E1 -24600.981,E2 -24600.981} C_VEL
LIN {X 0,Y 157.88,Z 443.327,A -85,B 0,C 180,E1 -24603.829,E2 -24603.829} C_VEL
LIN {X 0,Y 158.975,Z 436.718,A -85,B 0,C 180,E1 -24606.47,E2 -24606.47} C_VEL
LIN {X 0,Y 160.422,Z 432.262,A -85,B 0,C 180,E1 -24607.761,E2 -24607.761} C_VEL
LIN {X 0,Y 164.078,Z 423.186,A -85,B 0,C 180,E1 -24609.582,E2 -24609.582} C_VEL
LIN {X 0,Y 167.378,Z 413.575,A -85,B 0,C 180,E1 -24611,E2 -24611} C_VEL
LIN {X 0,Y 169.911,Z 404.376,A -85,B 0,C 180,E1 -24612.003,E2 -24612.003} C_VEL
LIN {X 0,Y 172.099,Z 393.379,A -85,B 0,C 180,E1 -24612.878,E2 -24612.878} C_VEL
LIN {X 0,Y 173.68,Z 379.074,A -85,B 0,C 180,E1 -24613.542,E2 -24613.542} C_VEL
LIN {X 0,Y 174.164,Z 372.002,A -85,B 0,C 180,E1 -24613.854,E2 -24613.854} C_VEL
LIN {X 0,Y 170.944,Z 363.175,A -85,B 0,C 180,E1 -24615.997,E2 -24615.997} C_VEL
LIN {X 0,Y 166.945,Z 354.255,A -85,B 0,C 180,E1 -24618.817,E2 -24618.817} C_VEL
LIN {X 0,Y 163.326,Z 347.454,A -85,B 0,C 180,E1 -24621.644,E2 -24621.644} C_VEL
LIN {X 0,Y 161.183,Z 343.723,A -85,B 0,C 180,E1 -24623.502,E2 -24623.502} C_VEL
LIN {X 0,Y 159.4,Z 340.85,A -85,B 0,C 180,E1 -24625.206,E2 -24625.206} C_VEL
LIN {X 0,Y 156.843,Z 337.465,A -85,B 0,C 180,E1 -24627.849,E2 -24627.849} C_VEL
LIN {X 0,Y 156.18,Z 336.361,A -85,B 0,C 180,E1 -24628.643,E2 -24628.643} C_VEL
LIN {X 0,Y 153.577,Z 333.439,A -85,B 0,C 180,E1 -24632.073,E2 -24632.073} C_VEL
LIN {X 0,Y 152.517,Z 331.275,A -85,B 0,C 180,E1 -24633.931,E2 -24633.931} C_VEL
LIN {X 0,Y 149.055,Z 327.701,A -85,B 0,C 180,E1 -24644.97,E2 -24644.97} C_VEL
LIN {X 0,Y 149.25,Z 327.638,A -85,B 0,C 180,E1 -24649.144,E2 -24649.144} C_VEL
LIN {X 0,Y 152.18,Z 330.675,A -85,B 0,C 180,E1 -24657.871,E2 -24657.871} C_VEL
LIN {X 0,Y 153.187,Z 331.414,A -85,B 0,C 180,E1 -24659.507,E2 -24659.507} C_VEL
LIN {X 0,Y 154.787,Z 334.557,A -85,B 0,C 180,E1 -24662.035,E2 -24662.035} C_VEL
LIN {X 0,Y 156.966,Z 336.87,A -85,B 0,C 180,E1 -24664.655,E2 -24664.655} C_VEL
LIN {X 0,Y 159.751,Z 340.757,A -85,B 0,C 180,E1 -24667.523,E2 -24667.523} C_VEL
LIN {X 0,Y 163.489,Z 346.599,A -85,B 0,C 180,E1 -24670.84,E2 -24670.84} C_VEL
LIN {X 0,Y 166.784,Z 351.753,A -85,B 0,C 180,E1 -24673.324,E2 -24673.324} C_VEL
LIN {X 0,Y 171.25,Z 359.408,A -85,B 0,C 180,E1 -24676.312,E2 -24676.312} C_VEL
LIN {X 0,Y 174.541,Z 366.155,A -85,B 0,C 180,E1 -24678.335,E2 -24678.335} C_VEL
LIN {X 0,Y 172.859,Z 384.739,A -85,B 0,C 180,E1 -24679.144,E2 -24679.144} C_VEL
LIN {X 0,Y 170.701,Z 397.187,A -85,B 0,C 180,E1 -24680.084,E2 -24680.084} C_VEL
LIN {X 0,Y 168.233,Z 407.155,A -85,B 0,C 180,E1 -24681.238,E2 -24681.238} C_VEL
LIN {X 0,Y 165.708,Z 415.145,A -85,B 0,C 180,E1 -24682.44,E2 -24682.44} C_VEL
LIN {X 0,Y 162.49,Z 423.459,A -85,B 0,C 180,E1 -24684.02,E2 -24684.02} C_VEL
LIN {X 0,Y 158.897,Z 431.547,A -85,B 0,C 180,E1 -24686.024,E2 -24686.024} C_VEL
LIN {X 0,Y 154.365,Z 440.133,A -85,B 0,C 180,E1 -24688.79,E2 -24688.79} C_VEL
LIN {X 0,Y 150.539,Z 446.277,A -85,B 0,C 180,E1 -24691.433,E2 -24691.433} C_VEL
LIN {X 0,Y 146.857,Z 451.53,A -85,B 0,C 180,E1 -24694.361,E2 -24694.361} C_VEL
LIN {X 0,Y 144.375,Z 454.931,A -85,B 0,C 180,E1 -24696.754,E2 -24696.754} C_VEL
LIN {X 0,Y 141.18,Z 458.74,A -85,B 0,C 180,E1 -24700.327,E2 -24700.327} C_VEL
LIN {X 0,Y 139.169,Z 460.853,A -85,B 0,C 180,E1 -24702.927,E2 -24702.927} C_VEL
LIN {X 0,Y 136.317,Z 463.362,A -85,B 0,C 180,E1 -24707.917,E2 -24707.917} C_VEL
LIN {X 0,Y 134.9,Z 464.245,A -85,B 0,C 180,E1 -24711.396,E2 -24711.396} C_VEL
LIN {X 0,Y 133.925,Z 464.466,A -85,B 0,C 180,E1 -24714.744,E2 -24714.744} C_VEL
LIN {X 0,Y 133.332,Z 464.027,A -85,B 0,C 180,E1 -24718.191,E2 -24718.191} C_VEL
LIN {X 0,Y 133.061,Z 462.92,A -85,B 0,C 180,E1 -24721.618,E2 -24721.618} C_VEL
LIN {X 0,Y 133.45,Z 460.012,A -85,B 0,C 180,E1 -24726.736,E2 -24726.736} C_VEL
LIN {X 0,Y 134.412,Z 455.581,A -85,B 0,C 180,E1 -24731.717,E2 -24731.717} C_VEL
LIN {X 0,Y 135.638,Z 450.654,A -85,B 0,C 180,E1 -24735.753,E2 -24735.753} C_VEL
LIN {X 0,Y 137.385,Z 444.322,A -85,B 0,C 180,E1 -24739.686,E2 -24739.686} C_VEL
LIN {X 0,Y 139.115,Z 437.963,A -85,B 0,C 180,E1 -24742.745,E2 -24742.745} C_VEL
LIN {X 0,Y 141.215,Z 430.101,A -85,B 0,C 180,E1 -24745.732,E2 -24745.732} C_VEL
LIN {X 0,Y 143,Z 423.036,A -85,B 0,C 180,E1 -24747.888,E2 -24747.888} C_VEL
LIN {X 0,Y 144.622,Z 415.959,A -85,B 0,C 180,E1 -24749.652,E2 -24749.652} C_VEL
LIN {X 0,Y 146.358,Z 407.246,A -85,B 0,C 180,E1 -24751.376,E2 -24751.376} C_VEL
LIN {X 0,Y 147.721,Z 398.449,A -85,B 0,C 180,E1 -24752.727,E2 -24752.727} C_VEL
LIN {X 0,Y 148.94,Z 388.714,A -85,B 0,C 180,E1 -24753.813,E2 -24753.813} C_VEL
LIN {X 0,Y 149.945,Z 377.254,A -85,B 0,C 180,E1 -24754.628,E2 -24754.628} C_VEL
LIN {X 0,Y 151.476,Z 346.914,A -85,B 0,C 180,E1 -24756.076,E2 -24756.076} C_VEL
LIN {X 0,Y 148.526,Z 337.642,A -85,B 0,C 180,E1 -24757.191,E2 -24757.191} C_VEL
LIN {X 0,Y 139.495,Z 319.579,A -85,B 0,C 180,E1 -24760.299,E2 -24760.299} C_VEL
LIN {X 0,Y 136.734,Z 314.388,A -85,B 0,C 180,E1 -24761.318,E2 -24761.318} C_VEL
LIN {X 0,Y 136.486,Z 313.28,A -85,B 0,C 180,E1 -24761.482,E2 -24761.482} C_VEL
LIN {X 0,Y 136.202,Z 313.324,A -85,B 0,C 180,E1 -24768.035,E2 -24768.035} C_VEL
LIN {X 0,Y 136.196,Z 313.298,A -85,B 0,C 180,E1 -24771.745,E2 -24771.745} C_VEL
LIN {X 0,Y 136.117,Z 313.348,A -85,B 0,C 180,E1 -24778.628,E2 -24778.628} C_VEL
LIN {X 0,Y 136.045,Z 313.347,A -85,B 0,C 180,E1 -24784.627,E2 -24784.627} C_VEL
LIN {X 0,Y 136.033,Z 313.35,A -85,B 0,C 180,E1 -24789.198,E2 -24789.198} C_VEL
LIN {X 0,Y 136.02,Z 313.337,A -85,B 0,C 180,E1 -24793.666,E2 -24793.666} C_VEL
LIN {X 0,Y 136.076,Z 313.348,A -85,B 0,C 180,E1 -24797.823,E2 -24797.823} C_VEL
LIN {X 0,Y 136.082,Z 313.336,A -85,B 0,C 180,E1 -24801.702,E2 -24801.702} C_VEL
LIN {X 0,Y 136.09,Z 313.319,A -85,B 0,C 180,E1 -24805.716,E2 -24805.716} C_VEL
LIN {X 0,Y 136.142,Z 313.338,A -85,B 0,C 180,E1 -24812.315,E2 -24812.315} C_VEL
LIN {X 0,Y 136.24,Z 313.294,A -85,B 0,C 180,E1 -24818.832,E2 -24818.832} C_VEL
LIN {X 0,Y 136.264,Z 313.322,A -85,B 0,C 180,E1 -24825.055,E2 -24825.055} C_VEL
LIN {X 0,Y 136.428,Z 313.303,A -85,B 0,C 180,E1 -24828.165,E2 -24828.165} C_VEL
LIN {X 0,Y 136.547,Z 313.277,A -85,B 0,C 180,E1 -24831.117,E2 -24831.117} C_VEL
LIN {X 0,Y 137.127,Z 313.211,A -85,B 0,C 180,E1 -24840,E2 -24840} C_VEL
LIN {X 0,Y 136.546,Z 313.264,A -85,B 0,C 180,E1 -24848.882,E2 -24848.882} C_VEL
LIN {X 0,Y 136.437,Z 313.288,A -85,B 0,C 180,E1 -24851.89,E2 -24851.89} C_VEL
LIN {X 0,Y 136.233,Z 313.323,A -85,B 0,C 180,E1 -24858.03,E2 -24858.03} C_VEL
LIN {X 0,Y 136.192,Z 313.315,A -85,B 0,C 180,E1 -24861.746,E2 -24861.746} C_VEL
LIN {X 0,Y 136.095,Z 313.339,A -85,B 0,C 180,E1 -24868.615,E2 -24868.615} C_VEL
LIN {X 0,Y 136.04,Z 313.355,A -85,B 0,C 180,E1 -24874.63,E2 -24874.63} C_VEL
LIN {X 0,Y 136.024,Z 313.33,A -85,B 0,C 180,E1 -24879.196,E2 -24879.196} C_VEL
LIN {X 0,Y 135.976,Z 313.347,A -85,B 0,C 180,E1 -24883.649,E2 -24883.649} C_VEL
LIN {X 0,Y 136.012,Z 313.355,A -85,B 0,C 180,E1 -24889.972,E2 -24889.972} C_VEL
LIN {X 0,Y 137.192,Z 316.45,A -85,B 0,C 180,E1 -24890.538,E2 -24890.538} C_VEL
LIN {X 0,Y 139.966,Z 321.402,A -85,B 0,C 180,E1 -24891.539,E2 -24891.539} C_VEL
LIN {X 0,Y 145.406,Z 335.003,A -85,B 0,C 180,E1 -24893.607,E2 -24893.607} C_VEL
LIN {X 0,Y 148.723,Z 345.145,A -85,B 0,C 180,E1 -24894.891,E2 -24894.891} C_VEL
LIN {X 0,Y 150.668,Z 366.289,A -85,B 0,C 180,E1 -24896.477,E2 -24896.477} C_VEL
LIN {X 0,Y 149.323,Z 390.4,A -85,B 0,C 180,E1 -24897.716,E2 -24897.716} C_VEL
LIN {X 0,Y 147.995,Z 401.828,A -85,B 0,C 180,E1 -24898.705,E2 -24898.705} C_VEL
LIN {X 0,Y 146.285,Z 412.1,A -85,B 0,C 180,E1 -24900.099,E2 -24900.099} C_VEL
LIN {X 0,Y 144.745,Z 420.912,A -85,B 0,C 180,E1 -24901.745,E2 -24901.745} C_VEL
LIN {X 0,Y 142.638,Z 429.214,A -85,B 0,C 180,E1 -24903.677,E2 -24903.677} C_VEL
LIN {X 0,Y 140.755,Z 437.158,A -85,B 0,C 180,E1 -24906.067,E2 -24906.067} C_VEL
LIN {X 0,Y 138.972,Z 443.698,A -85,B 0,C 180,E1 -24908.492,E2 -24908.492} C_VEL
LIN {X 0,Y 137.242,Z 449.919,A -85,B 0,C 180,E1 -24911.334,E2 -24911.334} C_VEL
LIN {X 0,Y 135.895,Z 455.08,A -85,B 0,C 180,E1 -24914.246,E2 -24914.246} C_VEL
LIN {X 0,Y 134.666,Z 460.33,A -85,B 0,C 180,E1 -24917.951,E2 -24917.951} C_VEL
LIN {X 0,Y 133.768,Z 465.173,A -85,B 0,C 180,E1 -24922.453,E2 -24922.453} C_VEL
LIN {X 0,Y 133.485,Z 468.49,A -85,B 0,C 180,E1 -24926.982,E2 -24926.982} C_VEL
LIN {X 0,Y 133.534,Z 470.188,A -85,B 0,C 180,E1 -24930.339,E2 -24930.339} C_VEL
LIN {X 0,Y 133.461,Z 471.004,A -85,B 0,C 180,E1 -24933.018,E2 -24933.018} C_VEL
LIN {X 0,Y 133.57,Z 471.452,A -85,B 0,C 180,E1 -24936.04,E2 -24936.04} C_VEL
LIN {X 0,Y 133.989,Z 471.454,A -85,B 0,C 180,E1 -24939.053,E2 -24939.053} C_VEL
LIN {X 0,Y 134.73,Z 471.008,A -85,B 0,C 180,E1 -24942.043,E2 -24942.043} C_VEL
LIN {X 0,Y 135.829,Z 470.004,A -85,B 0,C 180,E1 -24944.993,E2 -24944.993} C_VEL
LIN {X 0,Y 138.09,Z 467.596,A -85,B 0,C 180,E1 -24949.318,E2 -24949.318} C_VEL
LIN {X 0,Y 141.113,Z 463.901,A -85,B 0,C 180,E1 -24953.479,E2 -24953.479} C_VEL
LIN {X 0,Y 143.679,Z 460.764,A -85,B 0,C 180,E1 -24956.118,E2 -24956.118} C_VEL
LIN {X 0,Y 147.264,Z 455.799,A -85,B 0,C 180,E1 -24959.285,E2 -24959.285} C_VEL
LIN {X 0,Y 151.278,Z 449.585,A -85,B 0,C 180,E1 -24962.293,E2 -24962.293} C_VEL
LIN {X 0,Y 154.775,Z 443.544,A -85,B 0,C 180,E1 -24964.582,E2 -24964.582} C_VEL
LIN {X 0,Y 157.407,Z 438.475,A -85,B 0,C 180,E1 -24966.185,E2 -24966.185} C_VEL
LIN {X 0,Y 160.422,Z 432.262,A -85,B 0,C 180,E1 -24967.761,E2 -24967.761} C_VEL
LIN {X 0,Y 161.875,Z 427.614,A -85,B 0,C 180,E1 -24968.968,E2 -24968.968} C_VEL
LIN {X 0,Y 162.981,Z 419.845,A -85,B 0,C 180,E1 -24971.122,E2 -24971.122} C_VEL
LIN {X 0,Y 163.924,Z 411.607,A -85,B 0,C 180,E1 -24972.989,E2 -24972.989} C_VEL
LIN {X 0,Y 165.005,Z 406.242,A -85,B 0,C 180,E1 -24973.73,E2 -24973.73} C_VEL
LIN {X 0,Y 167.14,Z 396.738,A -85,B 0,C 180,E1 -24974.548,E2 -24974.548} C_VEL
LIN {X 0,Y 168.678,Z 387.058,A -85,B 0,C 180,E1 -24975.096,E2 -24975.096} C_VEL
LIN {X 0,Y 169.758,Z 374.351,A -85,B 0,C 180,E1 -24975.677,E2 -24975.677} C_VEL
LIN {X 0,Y 166.643,Z 365.804,A -85,B 0,C 180,E1 -24977.958,E2 -24977.958} C_VEL
LIN {X 0,Y 163.248,Z 358.292,A -85,B 0,C 180,E1 -24980.623,E2 -24980.623} C_VEL
LIN {X 0,Y 159.905,Z 351.494,A -85,B 0,C 180,E1 -24983.576,E2 -24983.576} C_VEL
LIN {X 0,Y 157.409,Z 347.264,A -85,B 0,C 180,E1 -24986.059,E2 -24986.059} C_VEL
LIN {X 0,Y 154.858,Z 343.631,A -85,B 0,C 180,E1 -24988.917,E2 -24988.917} C_VEL
LIN {X 0,Y 151.562,Z 339.133,A -85,B 0,C 180,E1 -24993.702,E2 -24993.702} C_VEL
LIN {X 0,Y 151.05,Z 338.116,A -85,B 0,C 180,E1 -24994.718,E2 -24994.718} C_VEL
LIN {X 0,Y 148.09,Z 334.784,A -85,B 0,C 180,E1 -25004.87,E2 -25004.87} C_VEL
LIN {X 0,Y 148.056,Z 334.541,A -85,B 0,C 180,E1 -25006.271,E2 -25006.271} C_VEL
LIN {X 0,Y 148.38,Z 334.936,A -85,B 0,C 180,E1 -25009.923,E2 -25009.923} C_VEL
LIN {X 0,Y 151.181,Z 337.716,A -85,B 0,C 180,E1 -25017.857,E2 -25017.857} C_VEL
LIN {X 0,Y 151.714,Z 338.256,A -85,B 0,C 180,E1 -25018.813,E2 -25018.813} C_VEL
LIN {X 0,Y 153.652,Z 341.778,A -85,B 0,C 180,E1 -25021.926,E2 -25021.926} C_VEL
LIN {X 0,Y 155.218,Z 343.526,A -85,B 0,C 180,E1 -25023.895,E2 -25023.895} C_VEL
LIN {X 0,Y 158.218,Z 348.108,A -85,B 0,C 180,E1 -25027.177,E2 -25027.177} C_VEL
LIN {X 0,Y 161.385,Z 353.196,A -85,B 0,C 180,E1 -25030.131,E2 -25030.131} C_VEL
LIN {X 0,Y 164.844,Z 358.881,A -85,B 0,C 180,E1 -25032.856,E2 -25032.856} C_VEL
LIN {X 0,Y 168.964,Z 366.603,A -85,B 0,C 180,E1 -25035.778,E2 -25035.778} C_VEL
LIN {X 0,Y 170.176,Z 369.329,A -85,B 0,C 180,E1 -25036.587,E2 -25036.587} C_VEL
LIN {X 0,Y 168.419,Z 386.229,A -85,B 0,C 180,E1 -25037.304,E2 -25037.304} C_VEL
LIN {X 0,Y 166.598,Z 396.358,A -85,B 0,C 180,E1 -25038.082,E2 -25038.082} C_VEL
LIN {X 0,Y 163.808,Z 407.098,A -85,B 0,C 180,E1 -25039.291,E2 -25039.291} C_VEL
LIN {X 0,Y 160.914,Z 415.866,A -85,B 0,C 180,E1 -25040.626,E2 -25040.626} C_VEL
LIN {X 0,Y 157.526,Z 424.129,A -85,B 0,C 180,E1 -25042.221,E2 -25042.221} C_VEL
LIN {X 0,Y 153.616,Z 432.376,A -85,B 0,C 180,E1 -25044.315,E2 -25044.315} C_VEL
LIN {X 0,Y 148.621,Z 441.094,A -85,B 0,C 180,E1 -25047.26,E2 -25047.26} C_VEL
LIN {X 0,Y 144.3,Z 447.484,A -85,B 0,C 180,E1 -25050.178,E2 -25050.178} C_VEL
LIN {X 0,Y 140.155,Z 452.93,A -85,B 0,C 180,E1 -25053.477,E2 -25053.477} C_VEL
LIN {X 0,Y 136.504,Z 457.279,A -85,B 0,C 180,E1 -25057.063,E2 -25057.063} C_VEL
LIN {X 0,Y 133.703,Z 460.174,A -85,B 0,C 180,E1 -25060.346,E2 -25060.346} C_VEL
LIN {X 0,Y 131.057,Z 462.543,A -85,B 0,C 180,E1 -25064.198,E2 -25064.198} C_VEL
LIN {X 0,Y 128.611,Z 464.26,A -85,B 0,C 180,E1 -25069.025,E2 -25069.025} C_VEL
LIN {X 0,Y 127.334,Z 464.652,A -85,B 0,C 180,E1 -25072.619,E2 -25072.619} C_VEL
LIN {X 0,Y 126.479,Z 464.375,A -85,B 0,C 180,E1 -25076.46,E2 -25076.46} C_VEL
LIN {X 0,Y 126.053,Z 463.516,A -85,B 0,C 180,E1 -25079.883,E2 -25079.883} C_VEL
LIN {X 0,Y 126.157,Z 461.062,A -85,B 0,C 180,E1 -25085.304,E2 -25085.304} C_VEL
LIN {X 0,Y 127.058,Z 456.961,A -85,B 0,C 180,E1 -25090.618,E2 -25090.618} C_VEL
LIN {X 0,Y 128.459,Z 451.273,A -85,B 0,C 180,E1 -25095.748,E2 -25095.748} C_VEL
LIN {X 0,Y 130.257,Z 445.043,A -85,B 0,C 180,E1 -25099.929,E2 -25099.929} C_VEL
LIN {X 0,Y 132.521,Z 437.043,A -85,B 0,C 180,E1 -25103.912,E2 -25103.912} C_VEL
LIN {X 0,Y 134.433,Z 430.228,A -85,B 0,C 180,E1 -25106.586,E2 -25106.586} C_VEL
LIN {X 0,Y 136.338,Z 422.959,A -85,B 0,C 180,E1 -25108.892,E2 -25108.892} C_VEL
LIN {X 0,Y 138.047,Z 415.818,A -85,B 0,C 180,E1 -25110.729,E2 -25110.729} C_VEL
LIN {X 0,Y 139.886,Z 407.01,A -85,B 0,C 180,E1 -25112.52,E2 -25112.52} C_VEL
LIN {X 0,Y 141.355,Z 397.555,A -85,B 0,C 180,E1 -25114.003,E2 -25114.003} C_VEL
LIN {X 0,Y 142.818,Z 385.602,A -85,B 0,C 180,E1 -25115.3,E2 -25115.3} C_VEL
LIN {X 0,Y 143.887,Z 371.105,A -85,B 0,C 180,E1 -25116.134,E2 -25116.134} C_VEL
LIN {X 0,Y 145.059,Z 348.29,A -85,B 0,C 180,E1 -25117.268,E2 -25117.268} C_VEL
LIN {X 0,Y 142.643,Z 340.594,A -85,B 0,C 180,E1 -25118.256,E2 -25118.256} C_VEL
LIN {X 0,Y 134.27,Z 323.766,A -85,B 0,C 180,E1 -25121.317,E2 -25121.317} C_VEL
LIN {X 0,Y 131.023,Z 318,A -85,B 0,C 180,E1 -25122.58,E2 -25122.58} C_VEL
LIN {X 0,Y 129.51,Z 315.331,A -85,B 0,C 180,E1 -25123.195,E2 -25123.195} C_VEL
LIN {X 0,Y 129.25,Z 314.183,A -85,B 0,C 180,E1 -25123.442,E2 -25123.442} C_VEL
LIN {X 0,Y 129.126,Z 314.194,A -85,B 0,C 180,E1 -25129.06,E2 -25129.06} C_VEL
LIN {X 0,Y 129.108,Z 314.182,A -85,B 0,C 180,E1 -25132.398,E2 -25132.398} C_VEL
LIN {X 0,Y 129.036,Z 314.228,A -85,B 0,C 180,E1 -25139.372,E2 -25139.372} C_VEL
LIN {X 0,Y 128.961,Z 314.231,A -85,B 0,C 180,E1 -25145.168,E2 -25145.168} C_VEL
LIN {X 0,Y 128.937,Z 314.223,A -85,B 0,C 180,E1 -25150.849,E2 -25150.849} C_VEL
LIN {X 0,Y 128.971,Z 314.224,A -85,B 0,C 180,E1 -25155.104,E2 -25155.104} C_VEL
LIN {X 0,Y 129.002,Z 314.226,A -85,B 0,C 180,E1 -25159.702,E2 -25159.702} C_VEL
LIN {X 0,Y 128.996,Z 314.2,A -85,B 0,C 180,E1 -25164.806,E2 -25164.806} C_VEL
LIN {X 0,Y 129.014,Z 314.225,A -85,B 0,C 180,E1 -25170.641,E2 -25170.641} C_VEL
LIN {X 0,Y 129.026,Z 314.22,A -85,B 0,C 180,E1 -25174.166,E2 -25174.166} C_VEL
LIN {X 0,Y 129.105,Z 314.187,A -85,B 0,C 180,E1 -25177.727,E2 -25177.727} C_VEL
LIN {X 0,Y 129.148,Z 314.181,A -85,B 0,C 180,E1 -25180.943,E2 -25180.943} C_VEL
LIN {X 0,Y 129.373,Z 314.181,A -85,B 0,C 180,E1 -25187.903,E2 -25187.903} C_VEL
LIN {X 0,Y 129.47,Z 314.16,A -85,B 0,C 180,E1 -25190.627,E2 -25190.627} C_VEL
LIN {X 0,Y 130.083,Z 314.089,A -85,B 0,C 180,E1 -25200,E2 -25200} C_VEL
LIN {X 0,Y 129.469,Z 314.144,A -85,B 0,C 180,E1 -25209.372,E2 -25209.372} C_VEL
LIN {X 0,Y 129.34,Z 314.177,A -85,B 0,C 180,E1 -25212.553,E2 -25212.553} C_VEL
LIN {X 0,Y 129.145,Z 314.201,A -85,B 0,C 180,E1 -25219.057,E2 -25219.057} C_VEL
LIN {X 0,Y 129.104,Z 314.2,A -85,B 0,C 180,E1 -25222.399,E2 -25222.399} C_VEL
LIN {X 0,Y 129.023,Z 314.226,A -85,B 0,C 180,E1 -25225.834,E2 -25225.834} C_VEL
LIN {X 0,Y 129.014,Z 314.218,A -85,B 0,C 180,E1 -25229.358,E2 -25229.358} C_VEL
LIN {X 0,Y 128.956,Z 314.236,A -85,B 0,C 180,E1 -25235.168,E2 -25235.168} C_VEL
LIN {X 0,Y 128.921,Z 314.206,A -85,B 0,C 180,E1 -25240.856,E2 -25240.856} C_VEL
LIN {X 0,Y 128.927,Z 314.236,A -85,B 0,C 180,E1 -25247.383,E2 -25247.383} C_VEL
LIN {X 0,Y 128.94,Z 314.235,A -85,B 0,C 180,E1 -25248.129,E2 -25248.129} C_VEL
LIN {X 0,Y 129.988,Z 317.181,A -85,B 0,C 180,E1 -25248.675,E2 -25248.675} C_VEL
LIN {X 0,Y 131.431,Z 319.551,A -85,B 0,C 180,E1 -25249.242,E2 -25249.242} C_VEL
LIN {X 0,Y 135.13,Z 326.466,A -85,B 0,C 180,E1 -25250.681,E2 -25250.681} C_VEL
LIN {X 0,Y 140.66,Z 341.058,A -85,B 0,C 180,E1 -25252.937,E2 -25252.937} C_VEL
LIN {X 0,Y 142.583,Z 347.501,A -85,B 0,C 180,E1 -25253.764,E2 -25253.764} C_VEL
LIN {X 0,Y 144.271,Z 366.994,A -85,B 0,C 180,E1 -25255.3,E2 -25255.3} C_VEL
